KUKA KRL program: MyProgram_020().src

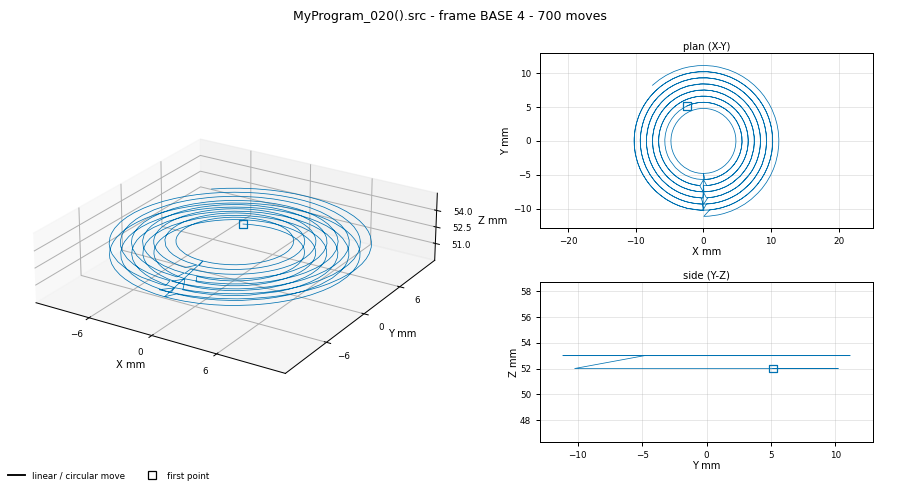
[picture p0: tool path of MyProgram_020().src in frame BASE 4, 700 of 700 moves have a stored position in this frame; points joined in program order, loops and branches not executed]
&ACCESS RVP
&REL 1
&PARAM TEMPLATE = C:\KRC\Roboter\Template\vorgabe
&PARAM EDITMASK = *
DEF MyProgram_020()
; ---- Setting reference (Base) ----
$BASE = BASE_DATA[4]

; --------------------------
; ---- Setting tool (TCP) ----
$TOOL = TOOL_DATA[3]
; --------------------------

$VEL.CP = VEL_APROX_PRINT
Startdeposition()
$VEL.CP = VEL_PRINT
LIN {X -2.4289,Y 5.1735,Z 52,A 107.8643,B 7.4449,C -0.6413,E1 7.4115,E2 338.3132} C_DIS
LIN {X -1.6441,Y 5.4719,Z 52,A 99.8653,B 7.4442,C -0.6489,E1 7.4326,E2 346.3058} C_DIS
LIN {X -0.8249,Y 5.6543,Z 52,A 90.902,B 7.4438,C -0.6532,E1 7.4572,E2 355.2666} C_DIS
LIN {X 0.0125,Y 5.7128,Z 52,A 82.6554,B 7.4438,C -0.654,E1 7.4801,E2 363.5085} C_DIS
LIN {X 0.8493,Y 5.6486,Z 52,A 74.2833,B 7.444,C -0.6514,E1 7.5034,E2 371.877} C_DIS
LIN {X 1.6675,Y 5.4622,Z 52,A 66.0095,B 7.4445,C -0.6455,E1 7.5257,E2 380.1475} C_DIS
LIN {X 2.45,Y 5.1592,Z 52,A 57.6846,B 7.4453,C -0.6363,E1 7.547,E2 388.4701} C_DIS
LIN {X 3.1799,Y 4.7453,Z 52,A 49.0733,B 7.4464,C -0.6235,E1 7.5674,E2 397.0811} C_DIS
LIN {X 3.84,Y 4.2269,Z 52,A 40.9883,B 7.4475,C -0.6091,E1 7.5847,E2 405.1642} C_DIS
LIN {X 4.4185,Y 3.6191,Z 52,A 32.7931,B 7.4489,C -0.5921,E1 7.5998,E2 413.359} C_DIS
LIN {X 4.9013,Y 2.9327,Z 52,A 24.252,B 7.4505,C -0.5719,E1 7.6128,E2 421.9018} C_DIS
LIN {X 5.2775,Y 2.1826,Z 52,A 16.2305,B 7.452,C -0.5517,E1 7.6221,E2 429.9236} C_DIS
LIN {X 5.5407,Y 1.3859,Z 52,A 7.7366,B 7.4536,C -0.5287,E1 7.6287,E2 438.4207} C_DIS
LIN {X 5.6841,Y 0.559,Z 52,A -0.2052,B 7.4552,C -0.5068,E1 7.6317,E2 446.3637} C_DIS
LIN {X 5.7063,Y -0.2799,Z 52,A -8.637,B 7.4567,C -0.483,E1 7.6315,E2 454.7997} C_DIS
LIN {X 5.6052,Y -1.1134,Z 52,A -14.4105,B 7.4577,C -0.4683,E1 7.6293,E2 460.5652} C_DIS
LIN {X 5.3986,Y -1.8885,Z 52,A -25.028,B 7.4595,C -0.4378,E1 7.621,E2 471.1999} C_DIS
LIN {X 5.0036,Y -2.7563,Z 52,A -33.9588,B 7.4608,C -0.4152,E1 7.61,E2 480.1335} C_DIS
LIN {X 4.593,Y -3.3992,Z 52,A -41.3661,B 7.4617,C -0.3977,E1 7.5983,E2 487.5447} C_DIS
LIN {X 4.0994,Y -3.9806,Z 52,A -49.0567,B 7.4626,C -0.3811,E1 7.5839,E2 495.2405} C_DIS
LIN {X 3.5319,Y -4.4901,Z 52,A -56.3617,B 7.4633,C -0.3674,E1 7.5683,E2 502.5489} C_DIS
LIN {X 2.9036,Y -4.9227,Z 52,A -64.2388,B 7.4639,C -0.3545,E1 7.5497,E2 510.4321} C_DIS
LIN {X 2.0463,Y -5.3406,Z 52,A -74.1091,B 7.4645,C -0.3422,E1 7.5245,E2 520.3099} C_DIS
LIN {X 1.0479,Y -5.6234,Z 52,A -84.1452,B 7.4648,C -0.3346,E1 7.4972,E2 530.3501} C_DIS
LIN {X 0.0063,Y -5.7151,Z 52,A -91.1459,B 7.4648,C -0.334,E1 7.4778,E2 537.3392} C_DIS
Enddeposition()
LIN {X 0.0063,Y -5.7151,Z 52,A -91.1459,B 7.4648,C -0.334,E1 7.4778,E2 537.3392} C_DIS
Startdeposition()
$VEL.CP = VEL_PRINT
LIN {X 0.5059,Y -6.5997,Z 52,A -88.5846,B 14.3606,C -1.1497,E1 14.4231,E2 533.3207} C_DIS
LIN {X 1.2106,Y -6.5077,Z 52,A -82.7819,B 14.3603,C -1.1527,E1 14.4391,E2 527.5162} C_DIS
LIN {X 1.9017,Y -6.3422,Z 52,A -76.5011,B 14.3599,C -1.1585,E1 14.456,E2 521.2307} C_DIS
LIN {X 2.57,Y -6.1008,Z 52,A -70.0036,B 14.3592,C -1.1667,E1 14.4729,E2 514.7265} C_DIS
LIN {X 3.2083,Y -5.7883,Z 52,A -64.1643,B 14.3586,C -1.175,E1 14.4874,E2 508.884} C_DIS
LIN {X 3.8105,Y -5.411,Z 52,A -58.3414,B 14.3578,C -1.1846,E1 14.5009,E2 503.0578} C_DIS
LIN {X 4.3704,Y -4.9735,Z 52,A -51.9483,B 14.3567,C -1.1974,E1 14.5147,E2 496.6579} C_DIS
LIN {X 4.8775,Y -4.4757,Z 52,A -45.8563,B 14.3557,C -1.2106,E1 14.5265,E2 490.5605} C_DIS
LIN {X 5.3296,Y -3.9273,Z 52,A -39.7457,B 14.3545,C -1.2251,E1 14.537,E2 484.4443} C_DIS
LIN {X 5.7197,Y -3.3333,Z 52,A -33.6906,B 14.3532,C -1.2403,E1 14.5459,E2 478.3839} C_DIS
LIN {X 6.0441,Y -2.7011,Z 52,A -27.6738,B 14.3518,C -1.2562,E1 14.5532,E2 472.3621} C_DIS
LIN {X 6.2999,Y -2.038,Z 52,A -21.6099,B 14.3504,C -1.2729,E1 14.5588,E2 466.2929} C_DIS
LIN {X 6.4828,Y -1.3513,Z 52,A -15.3375,B 14.3488,C -1.291,E1 14.5629,E2 460.0143} C_DIS
LIN {X 6.5887,Y -0.6485,Z 52,A -9.1544,B 14.3472,C -1.3089,E1 14.565,E2 453.8255} C_DIS
LIN {X 6.6197,Y 0.0616,Z 52,A -3.3981,B 14.3457,C -1.3251,E1 14.5652,E2 448.0663} C_DIS
LIN {X 6.575,Y 0.7709,Z 52,A 2.9779,B 14.3441,C -1.3437,E1 14.5636,E2 441.6843} C_DIS
LIN {X 6.4526,Y 1.4709,Z 52,A 8.8677,B 14.3426,C -1.36,E1 14.5604,E2 435.7915} C_DIS
LIN {X 6.2583,Y 2.1544,Z 52,A 14.9851,B 14.341,C -1.3766,E1 14.5552,E2 429.6704} C_DIS
LIN {X 5.9913,Y 2.8129,Z 52,A 21.1227,B 14.3395,C -1.3927,E1 14.5484,E2 423.5294} C_DIS
LIN {X 5.6548,Y 3.4389,Z 52,A 27.1939,B 14.3381,C -1.4075,E1 14.5399,E2 417.4557} C_DIS
LIN {X 5.2532,Y 4.0251,Z 52,A 32.9462,B 14.3368,C -1.4202,E1 14.5306,E2 411.7031} C_DIS
LIN {X 4.7937,Y 4.5673,Z 52,A 39.7226,B 14.3354,C -1.435,E1 14.5179,E2 404.9217} C_DIS
LIN {X 4.2744,Y 5.0525,Z 52,A 45.4975,B 14.3344,C -1.4453,E1 14.5058,E2 399.1475} C_DIS
LIN {X 3.7079,Y 5.4814,Z 52,A 51.459,B 14.3335,C -1.4546,E1 14.4923,E2 393.1864} C_DIS
LIN {X 3.1001,Y 5.8495,Z 52,A 57.6669,B 14.3326,C -1.4631,E1 14.4772,E2 386.9783} C_DIS
LIN {X 2.4551,Y 6.1484,Z 52,A 63.8557,B 14.332,C -1.4697,E1 14.4613,E2 380.79} C_DIS
LIN {X 1.7816,Y 6.3754,Z 52,A 70.1248,B 14.3315,C -1.4746,E1 14.4446,E2 374.5216} C_DIS
LIN {X 1.0876,Y 6.5283,Z 52,A 76.1758,B 14.3312,C -1.4773,E1 14.428,E2 368.473} C_DIS
LIN {X 0.3815,Y 6.6083,Z 52,A 82.1093,B 14.3312,C -1.478,E1 14.4115,E2 362.543} C_DIS
LIN {X -0.3292,Y 6.612,Z 52,A 88.3773,B 14.3312,C -1.4772,E1 14.3941,E2 356.2775} C_DIS
LIN {X -1.0362,Y 6.5401,Z 52,A 94.7434,B 14.3315,C -1.4745,E1 14.3765,E2 349.914} C_DIS
LIN {X -1.7309,Y 6.3897,Z 52,A 100.697,B 14.332,C -1.4697,E1 14.3603,E2 343.9653} C_DIS
LIN {X -2.406,Y 6.1677,Z 52,A 106.9909,B 14.3326,C -1.4632,E1 14.3438,E2 337.6751} C_DIS
LIN {X -3.0531,Y 5.874,Z 52,A 113.1471,B 14.3334,C -1.4549,E1 14.3284,E2 331.5237} C_DIS
LIN {X -3.6652,Y 5.513,Z 52,A 119.5582,B 14.3344,C -1.4448,E1 14.3132,E2 325.1167} C_DIS
LIN {X -4.2335,Y 5.0864,Z 52,A 125.4069,B 14.3355,C -1.4336,E1 14.3004,E2 319.2746} C_DIS
LIN {X -4.7554,Y 4.6042,Z 52,A 131.6596,B 14.3368,C -1.4206,E1 14.2879,E2 313.0271} C_DIS
LIN {X -5.2215,Y 4.0678,Z 52,A 138.0783,B 14.3382,C -1.4062,E1 14.2766,E2 306.6131} C_DIS
LIN {X -5.6279,Y 3.4848,Z 52,A 143.9789,B 14.3396,C -1.3913,E1 14.2675,E2 300.7194} C_DIS
LIN {X -5.9707,Y 2.8622,Z 52,A 150.3688,B 14.3412,C -1.3749,E1 14.2594,E2 294.3344} C_DIS
LIN {X -6.2429,Y 2.2057,Z 52,A 156.6547,B 14.3428,C -1.3578,E1 14.2531,E2 288.0535} C_DIS
LIN {X -6.443,Y 1.5238,Z 52,A 162.8172,B 14.3444,C -1.3404,E1 14.2487,E2 281.8967} C_DIS
LIN {X -6.5695,Y 0.8245,Z 52,A 169.0218,B 14.346,C -1.3226,E1 14.2461,E2 275.6972} C_DIS
LIN {X -6.6205,Y 0.1156,Z 52,A 175.3298,B 14.3476,C -1.3045,E1 14.2453,E2 269.3938} C_DIS
LIN {X -6.5942,Y -0.5946,Z 52,A -178.5062,B 14.3492,C -1.2868,E1 14.2464,E2 263.2346} C_DIS
LIN {X -6.493,Y -1.2981,Z 52,A -172.1603,B 14.3507,C -1.2691,E1 14.2494,E2 256.8923} C_DIS
LIN {X -6.3143,Y -1.9859,Z 52,A -165.8812,B 14.3522,C -1.252,E1 14.2543,E2 250.6166} C_DIS
LIN {X -6.0635,Y -2.6508,Z 52,A -159.9404,B 14.3535,C -1.2361,E1 14.2605,E2 244.6802} C_DIS
LIN {X -5.7462,Y -3.2866,Z 52,A -153.5703,B 14.3548,C -1.2205,E1 14.2689,E2 238.3123} C_DIS
LIN {X -5.3603,Y -3.8833,Z 52,A -147.4437,B 14.356,C -1.2063,E1 14.2786,E2 232.1883} C_DIS
LIN {X -4.9136,Y -4.4361,Z 52,A -141.2576,B 14.3571,C -1.1932,E1 14.2898,E2 226.004} C_DIS
LIN {X -4.4101,Y -4.9378,Z 52,A -134.9577,B 14.358,C -1.1815,E1 14.3026,E2 219.7047} C_DIS
LIN {X -3.8554,Y -5.382,Z 52,A -128.8622,B 14.3588,C -1.1715,E1 14.3162,E2 213.6102} C_DIS
LIN {X -3.2567,Y -5.7648,Z 52,A -122.6586,B 14.3595,C -1.163,E1 14.331,E2 207.4065} C_DIS
LIN {X -2.6196,Y -6.0793,Z 52,A -116.4199,B 14.36,C -1.1564,E1 14.3468,E2 201.1667} C_DIS
LIN {X -1.9529,Y -6.3257,Z 52,A -110.0034,B 14.3604,C -1.1517,E1 14.3638,E2 194.7477} C_DIS
LIN {X -1.2629,Y -6.4961,Z 52,A -104.1246,B 14.3606,C -1.1486,E1 14.3798,E2 188.8685} C_DIS
LIN {X -0.5594,Y -6.5953,Z 52,A -98.0781,B 14.3607,C -1.1473,E1 14.3966,E2 182.8202} C_DIS
LIN {X -0.5594,Y -6.5953,Z 52,A -98.0781,B 14.3607,C -1.1473,E1 14.3966,E2 182.8202} C_DIS
Enddeposition()
LIN {X -0.0274,Y -7.5244,Z 52,A -96.5126,B 21.2617,C -2.355,E1 21.386,E2 179.6143} C_DIS
Startdeposition()
$VEL.CP = VEL_PRINT
LIN {X -0.7814,Y -7.4872,Z 52,A -104.2237,B 21.2622,C -2.351,E1 21.3645,E2 187.3398} C_DIS
LIN {X -1.7575,Y -7.3207,Z 52,A -111.969,B 21.2619,C -2.3537,E1 21.3433,E2 195.0882} C_DIS
LIN {X -2.7152,Y -7.0156,Z 52,A -119.2275,B 21.2612,C -2.3604,E1 21.3242,E2 202.3448} C_DIS
LIN {X -3.4481,Y -6.6852,Z 52,A -125.2958,B 21.2604,C -2.3675,E1 21.309,E2 208.4122} C_DIS
LIN {X -4.1421,Y -6.2795,Z 52,A -131.442,B 21.2595,C -2.3762,E1 21.2944,E2 214.5574} C_DIS
LIN {X -4.7888,Y -5.8017,Z 52,A -137.6042,B 21.2584,C -2.3866,E1 21.2808,E2 220.7177} C_DIS
LIN {X -5.3803,Y -5.2573,Z 52,A -143.6754,B 21.2571,C -2.3986,E1 21.2687,E2 226.7856} C_DIS
LIN {X -6.0374,Y -4.4969,Z 52,A -151.9759,B 21.2552,C -2.4157,E1 21.2541,E2 235.0848} C_DIS
LIN {X -6.6618,Y -3.4963,Z 52,A -160.598,B 21.2528,C -2.4381,E1 21.242,E2 243.698} C_DIS
LIN {X -7.1224,Y -2.4411,Z 52,A -170.0178,B 21.2501,C -2.4625,E1 21.2324,E2 253.1129} C_DIS
LIN {X -7.3822,Y -1.4736,Z 52,A -177.4448,B 21.2477,C -2.4844,E1 21.2277,E2 260.5309} C_DIS
LIN {X -7.5117,Y -0.49,Z 52,A 175.1182,B 21.2452,C -2.5068,E1 21.2256,E2 267.9588} C_DIS
LIN {X -7.5011,Y 0.6008,Z 52,A 168.4839,B 21.2425,C -2.5302,E1 21.226,E2 274.5756} C_DIS
LIN {X -7.3321,Y 1.704,Z 52,A 157.0482,B 21.2393,C -2.5585,E1 21.2317,E2 286.0133} C_DIS
LIN {X -6.9123,Y 2.9745,Z 52,A 148.1141,B 21.236,C -2.5868,E1 21.2403,E2 294.929} C_DIS
LIN {X -6.3173,Y 4.0959,Z 52,A 138.4221,B 21.233,C -2.6128,E1 21.2537,E2 304.609} C_DIS
LIN {X -5.7816,Y 4.8207,Z 52,A 131.1882,B 21.2309,C -2.63,E1 21.2661,E2 311.8358} C_DIS
LIN {X -4.9317,Y 5.6867,Z 52,A 121.5646,B 21.2285,C -2.6503,E1 21.2855,E2 321.4502} C_DIS
LIN {X -3.9768,Y 6.3909,Z 52,A 112.154,B 21.2266,C -2.6668,E1 21.3072,E2 330.8528} C_DIS
LIN {X -3.1751,Y 6.826,Z 52,A 104.5371,B 21.2254,C -2.6765,E1 21.3263,E2 338.4661} C_DIS
LIN {X -1.7524,Y 7.3221,Z 52,A 94.415,B 21.2238,C -2.6895,E1 21.3533,E2 348.5726} C_DIS
LIN {X -0.7984,Y 7.4853,Z 52,A 87.1848,B 21.2233,C -2.694,E1 21.3732,E2 355.7973} C_DIS
LIN {X 0.1483,Y 7.5262,Z 52,A 79.6626,B 21.2232,C -2.6949,E1 21.3942,E2 363.3174} C_DIS
LIN {X 1.1941,Y 7.4322,Z 52,A 71.8258,B 21.2233,C -2.6936,E1 21.4159,E2 371.1506} C_DIS
LIN {X 2.1413,Y 7.2172,Z 52,A 64.1331,B 21.224,C -2.6884,E1 21.4367,E2 378.8437} C_DIS
LIN {X 3.0246,Y 6.8934,Z 52,A 56.7749,B 21.2249,C -2.6807,E1 21.4557,E2 386.2029} C_DIS
LIN {X 4.1385,Y 6.2822,Z 52,A 47.6638,B 21.2263,C -2.6693,E1 21.4776,E2 395.3123} C_DIS
LIN {X 4.7085,Y 5.8745,Z 52,A 41.823,B 21.2276,C -2.6581,E1 21.4905,E2 401.1581} C_DIS
LIN {X 5.57,Y 5.0582,Z 52,A 33.2892,B 21.2295,C -2.642,E1 21.5073,E2 409.6932} C_DIS
LIN {X 6.1111,Y 4.3879,Z 52,A 26.9308,B 21.2312,C -2.6278,E1 21.5181,E2 416.0546} C_DIS
LIN {X 6.715,Y 3.4036,Z 52,A 17.7733,B 21.234,C -2.6038,E1 21.5307,E2 425.2216} C_DIS
LIN {X 7.1416,Y 2.3681,Z 52,A 11.3801,B 21.2356,C -2.5907,E1 21.5373,E2 431.6086} C_DIS
LIN {X 7.3518,Y 1.6184,Z 52,A 3.4647,B 21.2387,C -2.5638,E1 21.5428,E2 439.5435} C_DIS
LIN {X 7.5047,Y 0.5929,Z 52,A -4.3405,B 21.2413,C -2.5408,E1 21.5454,E2 447.3571} C_DIS
LIN {X 7.5175,Y -0.4036,Z 52,A -11.7653,B 21.2438,C -2.5187,E1 21.545,E2 454.7899} C_DIS
LIN {X 7.4202,Y -1.2685,Z 52,A -19.3373,B 21.2466,C -2.494,E1 21.5418,E2 462.3766} C_DIS
LIN {X 7.0514,Y -2.6343,Z 52,A -28.9248,B 21.2495,C -2.4683,E1 21.5338,E2 471.9698} C_DIS
LIN {X 6.7153,Y -3.403,Z 52,A -35.7286,B 21.2517,C -2.4483,E1 21.5256,E2 478.7848} C_DIS
LIN {X 6.1358,Y -4.3568,Z 52,A -42.0446,B 21.253,C -2.4361,E1 21.5162,E2 485.0964} C_DIS
LIN {X 5.4535,Y -5.1882,Z 52,A -53.8238,B 21.2569,C -2.4006,E1 21.4945,E2 496.9101} C_DIS
LIN {X 4.3237,Y -6.1617,Z 52,A -63.1188,B 21.2584,C -2.386,E1 21.4741,E2 506.2042} C_DIS
LIN {X 3.4446,Y -6.6892,Z 52,A -70.8047,B 21.2598,C -2.3735,E1 21.4555,E2 513.8971} C_DIS
LIN {X 2.4008,Y -7.136,Z 52,A -79.8175,B 21.2611,C -2.3612,E1 21.432,E2 522.9202} C_DIS
LIN {X 1.5119,Y -7.3741,Z 52,A -86.7893,B 21.2617,C -2.3551,E1 21.413,E2 529.897} C_DIS
LIN {X 0.7619,Y -7.4894,Z 52,A -92.7274,B 21.2621,C -2.3515,E1 21.3966,E2 535.8397} C_DIS
LIN {X -0.0274,Y -7.5244,Z 52,A -96.5127,B 21.2617,C -2.355,E1 21.386,E2 539.6144} C_DIS
Enddeposition()
LIN {X -0.0274,Y -7.5244,Z 52,A -96.5127,B 21.2617,C -2.355,E1 21.386,E2 539.6144} C_DIS
Startdeposition()
$VEL.CP = VEL_PRINT
LIN {X 0.4505,Y -8.4164,Z 52,A -93.4741,B 24.8134,C -3.1503,E1 25.0114,E2 535.6406} C_DIS
LIN {X 1.5174,Y -8.2959,Z 52,A -85.4803,B 24.8125,C -3.1575,E1 25.0336,E2 527.6369} C_DIS
LIN {X 2.6389,Y -8.0045,Z 52,A -77.6649,B 24.8115,C -3.1657,E1 25.0546,E2 519.8149} C_DIS
LIN {X 3.713,Y -7.57,Z 52,A -69.6264,B 24.8101,C -3.1779,E1 25.0751,E2 511.7673} C_DIS
LIN {X 4.7012,Y -7.0001,Z 52,A -62.0699,B 24.8085,C -3.1911,E1 25.093,E2 504.2033} C_DIS
LIN {X 5.435,Y -6.4462,Z 52,A -53.1824,B 24.8052,C -3.2179,E1 25.1121,E2 495.2863} C_DIS
LIN {X 7.0088,Y -4.6885,Z 52,A -40.2537,B 24.8023,C -3.2418,E1 25.1348,E2 482.361} C_DIS
LIN {X 7.4731,Y -3.9082,Z 52,A -33.7544,B 24.8,C -3.2609,E1 25.1437,E2 475.8499} C_DIS
LIN {X 7.8918,Y -2.9691,Z 52,A -26.4626,B 24.7972,C -3.2833,E1 25.1514,E2 468.5453} C_DIS
LIN {X 8.222,Y -1.8731,Z 52,A -18.8386,B 24.7944,C -3.3061,E1 25.1569,E2 460.9111} C_DIS
LIN {X 8.3909,Y -0.8376,Z 52,A -12.2741,B 24.792,C -3.3249,E1 25.1593,E2 454.3408} C_DIS
LIN {X 8.4309,Y 0.142,Z 52,A -5.498,B 24.7893,C -3.3462,E1 25.1596,E2 447.5544} C_DIS
LIN {X 8.3647,Y 1.0691,Z 52,A 1.2925,B 24.7865,C -3.3683,E1 25.1577,E2 440.7516} C_DIS
LIN {X 8.1134,Y 2.2842,Z 52,A 9.2044,B 24.7837,C -3.3904,E1 25.1526,E2 432.8332} C_DIS
LIN {X 7.7187,Y 3.3947,Z 52,A 17.3327,B 24.7807,C -3.4135,E1 25.1443,E2 424.6951} C_DIS
LIN {X 7.2312,Y 4.3372,Z 52,A 24.5613,B 24.7783,C -3.4324,E1 25.1345,E2 417.4593} C_DIS
LIN {X 6.6288,Y 5.2057,Z 52,A 31.6279,B 24.7761,C -3.4489,E1 25.1228,E2 410.3876} C_DIS
LIN {X 6.0725,Y 5.8426,Z 52,A 37.0713,B 24.7747,C -3.4598,E1 25.1126,E2 404.9424} C_DIS
LIN {X 5.4563,Y 6.4214,Z 52,A 42.825,B 24.7733,C -3.4708,E1 25.1006,E2 399.1853} C_DIS
LIN {X 4.6138,Y 7.0597,Z 52,A 50.4541,B 24.7715,C -3.4843,E1 25.0831,E2 391.5506} C_DIS
LIN {X 3.5901,Y 7.625,Z 52,A 57.9991,B 24.7704,C -3.4927,E1 25.0645,E2 384.0065} C_DIS
LIN {X 2.785,Y 7.9551,Z 52,A 63.8459,B 24.7697,C -3.4978,E1 25.0492,E2 378.1601} C_DIS
LIN {X 1.95,Y 8.1997,Z 52,A 69.7666,B 24.7692,C -3.5015,E1 25.0332,E2 372.24} C_DIS
LIN {X 0.7662,Y 8.3987,Z 52,A 78.3807,B 24.7688,C -3.5045,E1 25.0094,E2 363.6258} C_DIS
LIN {X -0.4208,Y 8.4227,Z 52,A 87.5718,B 24.7687,C -3.5053,E1 24.9838,E2 354.432} C_DIS
LIN {X -2.3301,Y 8.1054,Z 52,A 99.4928,B 24.7705,C -3.492,E1 24.9513,E2 342.5286} C_DIS
LIN {X -3.4977,Y 7.6741,Z 52,A 108.1812,B 24.7719,C -3.4809,E1 24.9289,E2 333.8473} C_DIS
LIN {X -4.5027,Y 7.1259,Z 52,A 115.3498,B 24.7737,C -3.467,E1 24.9116,E2 326.6906} C_DIS
LIN {X -5.4177,Y 6.461,Z 52,A 123.1877,B 24.7758,C -3.4514,E1 24.8942,E2 318.8616} C_DIS
LIN {X -6.1286,Y 5.7846,Z 52,A 129.6137,B 24.7778,C -3.436,E1 24.8815,E2 312.4455} C_DIS
LIN {X -6.8592,Y 4.9051,Z 52,A 137.784,B 24.7804,C -3.4162,E1 24.8674,E2 304.2843} C_DIS
LIN {X -7.5549,Y 3.7442,Z 52,A 147.3187,B 24.7837,C -3.3905,E1 24.8544,E2 294.7612} C_DIS
LIN {X -8.127,Y 2.2469,Z 52,A 160.9266,B 24.7879,C -3.3573,E1 24.8428,E2 281.1551} C_DIS
LIN {X -8.4128,Y 0.5678,Z 52,A 169.886,B 24.7924,C -3.3222,E1 24.8399,E2 272.2265} C_DIS
LIN {X -8.4247,Y -0.3871,Z 52,A 176.7329,B 24.7949,C -3.302,E1 24.8403,E2 265.3867} C_DIS
LIN {X -8.2786,Y -1.5841,Z 52,A -176.9993,B 24.7979,C -3.2777,E1 24.8426,E2 259.1397} C_DIS
LIN {X -8.1045,Y -2.3329,Z 52,A -169.8712,B 24.7999,C -3.2619,E1 24.8476,E2 252.008} C_DIS
LIN {X -7.751,Y -3.3079,Z 52,A -163.2341,B 24.8023,C -3.2422,E1 24.8542,E2 245.3808} C_DIS
LIN {X -7.3886,Y -4.054,Z 52,A -157.4386,B 24.8041,C -3.2273,E1 24.8617,E2 239.5901} C_DIS
LIN {X -6.8394,Y -4.9337,Z 52,A -149.9463,B 24.8062,C -3.2101,E1 24.8733,E2 232.1017} C_DIS
LIN {X -6.1425,Y -5.7759,Z 52,A -142.8279,B 24.8082,C -3.1937,E1 24.8864,E2 224.9904} C_DIS
LIN {X -5.3899,Y -6.4771,Z 52,A -136.0085,B 24.8098,C -3.1804,E1 24.9006,E2 218.1758} C_DIS
LIN {X -4.5644,Y -7.0908,Z 52,A -128.4213,B 24.811,C -3.1699,E1 24.918,E2 210.5878} C_DIS
LIN {X -3.6707,Y -7.5906,Z 52,A -121.6991,B 24.8121,C -3.161,E1 24.9346,E2 203.8685} C_DIS
LIN {X -2.7148,Y -7.9848,Z 52,A -114.2313,B 24.8127,C -3.1557,E1 24.9542,E2 196.3979} C_DIS
LIN {X -1.5311,Y -8.2879,Z 52,A -106.4733,B 24.8133,C -3.1506,E1 24.9753,E2 188.6421} C_DIS
LIN {X -0.3286,Y -8.4268,Z 52,A -98.0691,B 24.8133,C -3.1508,E1 24.9986,E2 180.2337} C_DIS
LIN {X -0.3286,Y -8.4268,Z 52,A -98.0691,B 24.8133,C -3.1508,E1 24.9986,E2 180.2337} C_DIS
Enddeposition()
LIN {X -0.052,Y -9.3359,Z 52,A -98.3791,B 24.8159,C -3.1288,E1 24.9976,E2 180.5961} C_DIS
Startdeposition()
$VEL.CP = VEL_PRINT
LIN {X -0.8395,Y -9.3001,Z 52,A -104.3026,B 24.8163,C -3.1254,E1 24.9811,E2 186.5298} C_DIS
LIN {X -1.9855,Y -9.1183,Z 52,A -111.0179,B 24.8159,C -3.1289,E1 24.9627,E2 193.2436} C_DIS
LIN {X -2.7999,Y -8.9013,Z 52,A -116.1132,B 24.8155,C -3.1324,E1 24.949,E2 198.3387} C_DIS
LIN {X -3.5922,Y -8.6137,Z 52,A -121.2417,B 24.8149,C -3.1372,E1 24.9357,E2 203.4669} C_DIS
LIN {X -4.6382,Y -8.1037,Z 52,A -128.6231,B 24.814,C -3.1455,E1 24.9174,E2 210.8486} C_DIS
LIN {X -5.456,Y -7.5777,Z 52,A -134.7044,B 24.8129,C -3.1546,E1 24.9033,E2 216.9285} C_DIS
LIN {X -6.282,Y -6.9086,Z 52,A -142.2,B 24.8115,C -3.1658,E1 24.8875,E2 224.4268} C_DIS
LIN {X -7.0554,Y -6.1139,Z 52,A -148.6364,B 24.8097,C -3.1807,E1 24.8755,E2 230.856} C_DIS
LIN {X -7.8689,Y -5.0191,Z 52,A -156.4687,B 24.8073,C -3.2012,E1 24.863,E2 238.6777} C_DIS
LIN {X -8.4491,Y -3.9729,Z 52,A -163.7812,B 24.8049,C -3.2206,E1 24.8535,E2 245.9827} C_DIS
LIN {X -8.7989,Y -3.1225,Z 52,A -169.5115,B 24.803,C -3.2364,E1 24.8478,E2 251.7073} C_DIS
LIN {X -9.0977,Y -2.0829,Z 52,A -176.1379,B 24.8006,C -3.256,E1 24.8431,E2 258.3253} C_DIS
LIN {X -9.2807,Y -1.0169,Z 52,A 177.0006,B 24.7981,C -3.2761,E1 24.8403,E2 265.1795} C_DIS
LIN {X -9.3371,Y 0.0703,Z 52,A 169.9229,B 24.7955,C -3.2968,E1 24.8399,E2 272.2501} C_DIS
LIN {X -9.269,Y 1.1202,Z 52,A 162.711,B 24.793,C -3.317,E1 24.8419,E2 279.4569} C_DIS
LIN {X -8.9578,Y 2.6352,Z 52,A 154.006,B 24.7894,C -3.3458,E1 24.8477,E2 288.1436} C_DIS
LIN {X -8.5926,Y 3.6417,Z 52,A 147.8018,B 24.7869,C -3.3653,E1 24.8539,E2 294.3359} C_DIS
LIN {X -8.1226,Y 4.6038,Z 52,A 140.5918,B 24.7845,C -3.3838,E1 24.8633,E2 301.5399} C_DIS
LIN {X -7.3654,Y 5.7368,Z 52,A 132.4678,B 24.7817,C -3.4059,E1 24.8764,E2 309.6507} C_DIS
LIN {X -6.6986,Y 6.5035,Z 52,A 126.1589,B 24.7798,C -3.4209,E1 24.8883,E2 315.9515} C_DIS
LIN {X -5.7812,Y 7.3262,Z 52,A 118.7773,B 24.7776,C -3.4374,E1 24.9039,E2 323.3221} C_DIS
LIN {X -5.0269,Y 7.8637,Z 52,A 112.9356,B 24.7762,C -3.448,E1 24.9174,E2 329.158} C_DIS
LIN {X -4.016,Y 8.4282,Z 52,A 105.736,B 24.7748,C -3.4592,E1 24.9352,E2 336.3506} C_DIS
LIN {X -2.9275,Y 8.8627,Z 52,A 98.7091,B 24.7735,C -3.4686,E1 24.9535,E2 343.3694} C_DIS
LIN {X -1.7907,Y 9.1636,Z 52,A 91.1938,B 24.7728,C -3.4744,E1 24.9739,E2 350.8809} C_DIS
LIN {X -0.6773,Y 9.3118,Z 52,A 84.2906,B 24.7723,C -3.4779,E1 24.9931,E2 357.7797} C_DIS
LIN {X 0.6229,Y 9.3154,Z 52,A 76.4024,B 24.7722,C -3.4791,E1 25.0151,E2 365.6637} C_DIS
LIN {X 1.7844,Y 9.1611,Z 52,A 69.2149,B 24.7724,C -3.4771,E1 25.0349,E2 372.849} C_DIS
LIN {X 2.6524,Y 8.9468,Z 52,A 63.9703,B 24.7728,C -3.4746,E1 25.049,E2 378.0913} C_DIS
LIN {X 3.7043,Y 8.5697,Z 52,A 56.8714,B 24.7737,C -3.4671,E1 25.0675,E2 385.1923} C_DIS
LIN {X 4.7988,Y 8.0048,Z 52,A 50.9112,B 24.7741,C -3.4643,E1 25.0822,E2 391.1423} C_DIS
LIN {X 5.4668,Y 7.5701,Z 52,A 44.5238,B 24.776,C -3.4498,E1 25.097,E2 397.5428} C_DIS
LIN {X 6.1655,Y 7.0114,Z 52,A 38.9428,B 24.7774,C -3.4392,E1 25.1089,E2 403.1274} C_DIS
LIN {X 7.152,Y 6.0011,Z 52,A 30.3335,B 24.7797,C -3.421,E1 25.1252,E2 411.7421} C_DIS
LIN {X 7.7543,Y 5.2005,Z 52,A 24.2516,B 24.7816,C -3.4066,E1 25.1351,E2 417.8287} C_DIS
LIN {X 8.3413,Y 4.186,Z 52,A 17.2885,B 24.7839,C -3.3891,E1 25.1445,E2 424.7969} C_DIS
LIN {X 8.8069,Y 3.1008,Z 52,A 10.0363,B 24.7865,C -3.3687,E1 25.1519,E2 432.0574} C_DIS
LIN {X 9.0454,Y 2.3117,Z 52,A 4.8737,B 24.7884,C -3.3533,E1 25.1558,E2 437.2269} C_DIS
LIN {X 9.2553,Y 1.2386,Z 52,A -3.0125,B 24.7919,C -3.326,E1 25.1592,E2 445.1317} C_DIS
LIN {X 9.3328,Y -0.2628,Z 52,A -10.8383,B 24.7944,C -3.3059,E1 25.1596,E2 452.9586} C_DIS
LIN {X 9.1482,Y -1.8645,Z 52,A -22.7728,B 24.7997,C -3.2631,E1 25.1543,E2 464.9245} C_DIS
LIN {X 8.6526,Y -3.5093,Z 52,A -31.0236,B 24.8019,C -3.245,E1 25.1468,E2 473.1717} C_DIS
LIN {X 8.0666,Y -4.704,Z 52,A -40.3815,B 24.8056,C -3.215,E1 25.1345,E2 482.5516} C_DIS
LIN {X 7.3945,Y -5.6982,Z 52,A -45.3651,B 24.8064,C -3.2088,E1 25.1265,E2 487.5255} C_DIS
LIN {X 6.7537,Y -6.4454,Z 52,A -54.3373,B 24.81,C -3.1782,E1 25.1096,E2 496.5306} C_DIS
LIN {X 5.4355,Y -7.5868,Z 52,A -61.872,B 24.8108,C -3.1716,E1 25.0934,E2 504.0525} C_DIS
LIN {X 4.8099,Y -8.0022,Z 52,A -68.0282,B 24.8128,C -3.1554,E1 25.0789,E2 510.2271} C_DIS
LIN {X 3.7305,Y -8.5544,Z 52,A -75.1902,B 24.814,C -3.1452,E1 25.0609,E2 517.3946} C_DIS
LIN {X 2.6834,Y -8.9427,Z 52,A -82.1917,B 24.8151,C -3.1362,E1 25.0423,E2 524.4037} C_DIS
LIN {X 1.6599,Y -9.189,Z 52,A -89.4964,B 24.8161,C -3.1275,E1 25.0223,E2 531.7201} C_DIS
LIN {X 0.4404,Y -9.323,Z 52,A -95.5715,B 24.8159,C -3.1289,E1 25.0055,E2 537.7885} C_DIS
LIN {X 0.4404,Y -9.323,Z 52,A -95.5715,B 24.8159,C -3.1289,E1 25.0055,E2 537.7885} C_DIS
Enddeposition()
LIN {X -0.0612,Y -10.2374,Z 52,A -97.9695,B 24.8176,C -3.1145,E1 24.9987,E2 540.2205} C_DIS
Startdeposition()
$VEL.CP = VEL_PRINT
LIN {X 0.6871,Y -10.2175,Z 52,A -92.1264,B 24.8167,C -3.1221,E1 25.015,E2 534.3609} C_DIS
LIN {X 1.7113,Y -10.0968,Z 52,A -86.2358,B 24.8162,C -3.1264,E1 25.0313,E2 528.4653} C_DIS
LIN {X 2.8814,Y -9.8282,Z 52,A -79.7051,B 24.8155,C -3.1323,E1 25.049,E2 521.9307} C_DIS
LIN {X 3.9668,Y -9.4385,Z 52,A -73.3076,B 24.8145,C -3.1406,E1 25.0657,E2 515.5273} C_DIS
LIN {X 4.8,Y -9.0423,Z 52,A -68.1956,B 24.8136,C -3.1486,E1 25.0784,E2 510.4101} C_DIS
LIN {X 5.5946,Y -8.5734,Z 52,A -63.1215,B 24.8125,C -3.1576,E1 25.0905,E2 505.3309} C_DIS
LIN {X 6.6386,Y -7.7967,Z 52,A -55.8131,B 24.8107,C -3.1729,E1 25.1065,E2 498.0132} C_DIS
LIN {X 7.4442,Y -7.0269,Z 52,A -49.6235,B 24.809,C -3.1873,E1 25.1188,E2 491.8155} C_DIS
LIN {X 8.0272,Y -6.3523,Z 52,A -44.7338,B 24.8075,C -3.1993,E1 25.1275,E2 486.9197} C_DIS
LIN {X 8.5502,Y -5.6302,Z 52,A -39.831,B 24.806,C -3.2121,E1 25.1353,E2 482.0107} C_DIS
LIN {X 9.0088,Y -4.8655,Z 52,A -34.8074,B 24.8042,C -3.2263,E1 25.1423,E2 476.9794} C_DIS
LIN {X 9.4867,Y -3.8588,Z 52,A -28.3755,B 24.8018,C -3.2457,E1 25.1495,E2 470.5366} C_DIS
LIN {X 9.8799,Y -2.6852,Z 52,A -22.9596,B 24.8005,C -3.257,E1 25.1542,E2 465.1245} C_DIS
LIN {X 10.0815,Y -1.8057,Z 52,A -16.4878,B 24.7974,C -3.2817,E1 25.158,E2 458.632} C_DIS
LIN {X 10.2129,Y -0.7557,Z 52,A -10.7283,B 24.7953,C -3.2991,E1 25.1596,E2 452.8653} C_DIS
LIN {X 10.2254,Y 0.5691,Z 52,A -3.0869,B 24.7922,C -3.3235,E1 25.1592,E2 445.2115} C_DIS
LIN {X 10.0787,Y 1.7954,Z 52,A 3.5193,B 24.7898,C -3.3426,E1 25.1566,E2 438.5989} C_DIS
LIN {X 9.8779,Y 2.6862,Z 52,A 8.5254,B 24.788,C -3.357,E1 25.1532,E2 433.5875} C_DIS
LIN {X 9.5994,Y 3.5558,Z 52,A 13.4788,B 24.7862,C -3.3707,E1 25.1487,E2 428.6296} C_DIS
LIN {X 9.2459,Y 4.3976,Z 52,A 18.7553,B 24.7843,C -3.3857,E1 25.1427,E2 423.3461} C_DIS
LIN {X 8.8161,Y 5.2032,Z 52,A 23.8601,B 24.7826,C -3.399,E1 25.1357,E2 418.2363} C_DIS
LIN {X 8.3163,Y 5.9674,Z 52,A 28.8739,B 24.7811,C -3.4109,E1 25.1277,E2 413.2188} C_DIS
LIN {X 7.7514,Y 6.6846,Z 52,A 33.8719,B 24.7796,C -3.4218,E1 25.1189,E2 408.2179} C_DIS
LIN {X 7.1257,Y 7.3495,Z 52,A 38.9606,B 24.7783,C -3.4323,E1 25.1089,E2 403.1261} C_DIS
LIN {X 6.4426,Y 7.9552,Z 52,A 44.1284,B 24.777,C -3.442,E1 25.0979,E2 397.9552} C_DIS
LIN {X 5.7087,Y 8.4984,Z 52,A 49.0874,B 24.776,C -3.4496,E1 25.0866,E2 392.9954} C_DIS
LIN {X 4.9289,Y 8.9734,Z 52,A 54.4375,B 24.775,C -3.4578,E1 25.0736,E2 387.6421} C_DIS
LIN {X 4.1092,Y 9.3757,Z 52,A 59.3893,B 24.7743,C -3.4628,E1 25.0611,E2 382.6908} C_DIS
LIN {X 3.2574,Y 9.7048,Z 52,A 64.455,B 24.7737,C -3.4671,E1 25.0478,E2 377.6254} C_DIS
LIN {X 2.3798,Y 9.9572,Z 52,A 69.5483,B 24.7733,C -3.47,E1 25.034,E2 372.533} C_DIS
LIN {X 1.7092,Y 10.0972,Z 52,A 74.0055,B 24.7729,C -3.4736,E1 25.0218,E2 368.0719} C_DIS
LIN {X 0.5608,Y 10.226,Z 52,A 80.5122,B 24.7729,C -3.4741,E1 25.0037,E2 361.5674} C_DIS
LIN {X -0.8075,Y 10.2063,Z 52,A 87.6056,B 24.7734,C -3.47,E1 24.9839,E2 354.4824} C_DIS
LIN {X -1.7266,Y 10.0914,Z 52,A 92.7707,B 24.7738,C -3.4666,E1 24.9697,E2 349.321} C_DIS
LIN {X -2.6317,Y 9.8943,Z 52,A 97.9163,B 24.7744,C -3.4618,E1 24.9557,E2 344.1799} C_DIS
LIN {X -3.5154,Y 9.6167,Z 52,A 103.2031,B 24.7752,C -3.4559,E1 24.9417,E2 338.8972} C_DIS
LIN {X -4.5793,Y 9.16,Z 52,A 110.1343,B 24.7763,C -3.4471,E1 24.9242,E2 331.9696} C_DIS
LIN {X -5.7429,Y 8.4765,Z 52,A 117.3701,B 24.7782,C -3.4331,E1 24.9071,E2 324.7446} C_DIS
LIN {X -6.4701,Y 7.933,Z 52,A 122.4181,B 24.7795,C -3.4226,E1 24.896,E2 319.7032} C_DIS
LIN {X -7.147,Y 7.328,Z 52,A 127.4329,B 24.781,C -3.4111,E1 24.8858,E2 314.6955} C_DIS
LIN {X -7.7686,Y 6.6665,Z 52,A 132.5126,B 24.7826,C -3.3987,E1 24.8763,E2 309.6228} C_DIS
LIN {X -8.3291,Y 5.9525,Z 52,A 137.7579,B 24.7843,C -3.3857,E1 24.8676,E2 304.3836} C_DIS
LIN {X -8.823,Y 5.1908,Z 52,A 142.6939,B 24.7861,C -3.3717,E1 24.8603,E2 299.4558} C_DIS
LIN {X -9.2496,Y 4.3896,Z 52,A 148.0022,B 24.7879,C -3.3573,E1 24.8537,E2 294.1537} C_DIS
LIN {X -9.6005,Y 3.5524,Z 52,A 153.0549,B 24.7898,C -3.3423,E1 24.8485,E2 289.1086} C_DIS
LIN {X -9.8773,Y 2.6878,Z 52,A 158.1339,B 24.7918,C -3.3269,E1 24.8445,E2 284.037} C_DIS
LIN {X -10.0771,Y 1.8023,Z 52,A 163.2087,B 24.7937,C -3.3113,E1 24.8417,E2 278.9697} C_DIS
LIN {X -10.198,Y 0.9025,Z 52,A 168.4066,B 24.7957,C -3.2956,E1 24.8401,E2 273.7785} C_DIS
LIN {X -10.2377,Y -0.0045,Z 52,A 173.5016,B 24.7976,C -3.2799,E1 24.8398,E2 268.6905} C_DIS
LIN {X -10.1972,Y -0.9115,Z 52,A 178.6629,B 24.7996,C -3.2643,E1 24.8408,E2 263.5356} C_DIS
LIN {X -10.0758,Y -1.8112,Z 52,A -176.2118,B 24.8015,C -3.2489,E1 24.843,E2 258.4166} C_DIS
LIN {X -9.8753,Y -2.6967,Z 52,A -171.1193,B 24.8033,C -3.2339,E1 24.8465,E2 253.3303} C_DIS
LIN {X -9.5976,Y -3.561,Z 52,A -166.1323,B 24.8051,C -3.2194,E1 24.851,E2 248.3498} C_DIS
LIN {X -9.2459,Y -4.3978,Z 52,A -160.8147,B 24.8067,C -3.2056,E1 24.8571,E2 243.0361} C_DIS
LIN {X -8.8187,Y -5.1988,Z 52,A -155.6812,B 24.8083,C -3.1925,E1 24.8641,E2 237.9071} C_DIS
LIN {X -8.3224,Y -5.9589,Z 52,A -150.8905,B 24.8099,C -3.1798,E1 24.8716,E2 233.1228} C_DIS
LIN {X -7.9126,Y -6.5029,Z 52,A -146.2833,B 24.8108,C -3.172,E1 24.8797,E2 228.5131} C_DIS
LIN {X -7.1244,Y -7.356,Z 52,A -140.2253,B 24.8125,C -3.158,E1 24.8915,E2 222.4625} C_DIS
LIN {X -6.3289,Y -8.0508,Z 52,A -134.4137,B 24.8138,C -3.1471,E1 24.9039,E2 216.6547} C_DIS
LIN {X -5.3658,Y -8.721,Z 52,A -129.0602,B 24.8152,C -3.1347,E1 24.9163,E2 211.3129} C_DIS
LIN {X -4.5747,Y -9.1622,Z 52,A -122.715,B 24.8157,C -3.1309,E1 24.9319,E2 204.959} C_DIS
LIN {X -3.5253,Y -9.6126,Z 52,A -116.3267,B 24.8164,C -3.1248,E1 24.9484,E2 198.571} C_DIS
LIN {X -2.3592,Y -9.9668,Z 52,A -109.2976,B 24.8168,C -3.1212,E1 24.9673,E2 191.5396} C_DIS
LIN {X -0.9586,Y -10.1972,Z 52,A -101.2361,B 24.817,C -3.12,E1 24.9896,E2 183.4746} C_DIS
LIN {X -0.0612,Y -10.2374,Z 52,A -97.9695,B 24.8176,C -3.1145,E1 24.9987,E2 180.2205} C_DIS
Enddeposition()
LIN {X 0.0024,Y -4.8127,Z 53,A -2.8481,B 0,C 0,E1 0.1598,E2 90.0716} C_DIS
Startdeposition()
$VEL.CP = VEL_PRINT
LIN {X -0.7063,Y -4.7565,Z 53,A -2.8719,B 0,C 0,E1 0.1598,E2 90.0717} C_DIS
LIN {X -1.2627,Y -4.6392,Z 53,A -2.8873,B 0,C 0,E1 0.1598,E2 90.0717} C_DIS
LIN {X -1.9345,Y -4.4065,Z 53,A -2.9021,B 0,C 0,E1 0.1598,E2 90.0717} C_DIS
LIN {X -2.82,Y -3.8913,Z 53,A -2.9125,B 0,C 0,E1 0.1598,E2 90.0715} C_DIS
LIN {X -3.3261,Y -3.47,Z 53,A -2.9132,B 0,C 0,E1 0.1598,E2 90.0715} C_DIS
LIN {X -3.7695,Y -2.983,Z 53,A -2.9088,B 0,C 0,E1 0.1598,E2 90.0715} C_DIS
LIN {X -4.1425,Y -2.44,Z 53,A -2.8994,B 0,C 0,E1 0.1598,E2 90.0715} C_DIS
LIN {X -4.4385,Y -1.8516,Z 53,A -2.8853,B 0,C 0,E1 0.1598,E2 90.0715} C_DIS
LIN {X -4.6474,Y -1.2269,Z 53,A -2.8664,B 0,C 0,E1 0.1598,E2 90.0715} C_DIS
LIN {X -4.7739,Y -0.5805,Z 53,A -2.8436,B 0,C 0,E1 0.1598,E2 90.0715} C_DIS
LIN {X -4.8062,Y 0.0773,Z 53,A -2.8168,B 0,C 0,E1 0.1598,E2 90.0715} C_DIS
LIN {X -4.7512,Y 0.7334,Z 53,A -2.7869,B 0,C 0,E1 0.1598,E2 90.0716} C_DIS
LIN {X -4.6063,Y 1.3759,Z 53,A -2.7544,B 0,C 0,E1 0.1598,E2 90.0716} C_DIS
LIN {X -4.375,Y 1.9926,Z 53,A -2.7197,B 0,C 0,E1 0.1598,E2 90.0717} C_DIS
LIN {X -4.0617,Y 2.5718,Z 53,A -2.6836,B 0,C 0,E1 0.1598,E2 90.0718} C_DIS
LIN {X -3.6727,Y 3.1034,Z 53,A -2.6467,B 0,C 0,E1 0.1598,E2 90.0718} C_DIS
LIN {X -3.2143,Y 3.5765,Z 53,A -2.6098,B 0,C 0,E1 0.1598,E2 90.072} C_DIS
LIN {X -2.6959,Y 3.983,Z 53,A -2.5735,B 0,C 0,E1 0.1598,E2 90.072} C_DIS
LIN {X -2.1259,Y 4.3136,Z 53,A -2.5385,B 0,C 0,E1 0.1598,E2 90.0721} C_DIS
LIN {X -1.5161,Y 4.5626,Z 53,A -2.5054,B 0,C 0,E1 0.1598,E2 90.0722} C_DIS
LIN {X -0.8781,Y 4.727,Z 53,A -2.475,B 0,C 0,E1 0.1598,E2 90.0722} C_DIS
LIN {X -0.2239,Y 4.8036,Z 53,A -2.4476,B 0,C 0,E1 0.1598,E2 90.0723} C_DIS
LIN {X 0.4347,Y 4.7894,Z 53,A -2.4239,B 0,C 0,E1 0.1598,E2 90.0723} C_DIS
LIN {X 1.0853,Y 4.6854,Z 53,A -2.4044,B 0,C 0,E1 0.1598,E2 90.0723} C_DIS
LIN {X 1.7154,Y 4.4932,Z 53,A -2.3893,B 0,C 0,E1 0.1598,E2 90.0723} C_DIS
LIN {X 2.3134,Y 4.2165,Z 53,A -2.379,B 0,C 0,E1 0.1598,E2 90.0723} C_DIS
LIN {X 2.8665,Y 3.8586,Z 53,A -2.3738,B 0,C 0,E1 0.1598,E2 90.0723} C_DIS
LIN {X 3.3672,Y 3.4308,Z 53,A -2.3736,B 0,C 0,E1 0.1598,E2 90.0723} C_DIS
LIN {X 3.805,Y 2.9388,Z 53,A -2.3784,B 0,C 0,E1 0.1598,E2 90.0723} C_DIS
LIN {X 4.1712,Y 2.3913,Z 53,A -2.3882,B 0,C 0,E1 0.1598,E2 90.0723} C_DIS
LIN {X 4.4594,Y 1.799,Z 53,A -2.4028,B 0,C 0,E1 0.1598,E2 90.0722} C_DIS
LIN {X 4.6646,Y 1.1729,Z 53,A -2.422,B 0,C 0,E1 0.1598,E2 90.0722} C_DIS
LIN {X 4.7809,Y 0.5244,Z 53,A -2.4453,B 0,C 0,E1 0.1598,E2 90.0721} C_DIS
LIN {X 4.8072,Y -0.1338,Z 53,A -2.4724,B 0,C 0,E1 0.1598,E2 90.0721} C_DIS
LIN {X 4.7431,Y -0.7894,Z 53,A -2.5028,B 0,C 0,E1 0.1598,E2 90.072} C_DIS
LIN {X 4.5908,Y -1.4303,Z 53,A -2.5357,B 0,C 0,E1 0.1598,E2 90.072} C_DIS
LIN {X 4.3507,Y -2.0437,Z 53,A -2.5708,B 0,C 0,E1 0.1598,E2 90.072} C_DIS
LIN {X 4.0313,Y -2.6197,Z 53,A -2.6071,B 0,C 0,E1 0.1598,E2 90.072} C_DIS
LIN {X 3.6341,Y -3.1451,Z 53,A -2.6442,B 0,C 0,E1 0.1598,E2 90.072} C_DIS
LIN {X 3.1722,Y -3.6146,Z 53,A -2.6812,B 0,C 0,E1 0.1598,E2 90.0719} C_DIS
LIN {X 2.6481,Y -4.0134,Z 53,A -2.7175,B 0,C 0,E1 0.1598,E2 90.0719} C_DIS
LIN {X 2.0742,Y -4.3369,Z 53,A -2.7524,B 0,C 0,E1 0.1598,E2 90.0719} C_DIS
LIN {X 1.462,Y -4.5798,Z 53,A -2.7852,B 0,C 0,E1 0.1598,E2 90.0719} C_DIS
LIN {X 0.8224,Y -4.7376,Z 53,A -2.8154,B 0,C 0,E1 0.1598,E2 90.0719} C_DIS
LIN {X 0.0024,Y -4.8127,Z 53,A -2.8487,B 0,C 0,E1 0.1598,E2 90.0718} C_DIS
Enddeposition()
LIN {X 0.0024,Y -4.8127,Z 53,A -2.8487,B 0,C 0,E1 0.1598,E2 90.0718} C_DIS
Startdeposition()
$VEL.CP = VEL_PRINT
LIN {X 0.2255,Y -5.7065,Z 53,A -88.058,B 6.4325,C -0.2436,E1 6.4504,E2 174.4545} C_DIS
LIN {X 1.0436,Y -5.6174,Z 53,A -79.6089,B 6.4323,C -0.2482,E1 6.4737,E2 166.0002} C_DIS
LIN {X 1.84,Y -5.4088,Z 53,A -71.3643,B 6.432,C -0.2558,E1 6.4958,E2 157.7511} C_DIS
LIN {X 2.5975,Y -5.087,Z 53,A -63.3868,B 6.4316,C -0.266,E1 6.516,E2 149.77} C_DIS
LIN {X 3.3026,Y -4.6626,Z 53,A -55.1183,B 6.431,C -0.2795,E1 6.5353,E2 141.4964} C_DIS
LIN {X 3.9376,Y -4.1388,Z 53,A -46.8352,B 6.4303,C -0.2957,E1 6.5526,E2 133.2079} C_DIS
LIN {X 4.4915,Y -3.53,Z 53,A -39.0387,B 6.4295,C -0.3127,E1 6.5666,E2 125.4086} C_DIS
LIN {X 4.9534,Y -2.8487,Z 53,A -32.9324,B 6.4288,C -0.3263,E1 6.5759,E2 119.308} C_DIS
LIN {X 5.347,Y -2.0255,Z 53,A -21.3288,B 6.4272,C -0.3577,E1 6.5891,E2 107.6872} C_DIS
LIN {X 5.6362,Y -0.9251,Z 53,A -10.6518,B 6.4255,C -0.3869,E1 6.5956,E2 97.0076} C_DIS
LIN {X 5.7102,Y -0.1171,Z 53,A -2.7563,B 6.4241,C -0.409,E1 6.5969,E2 89.1097} C_DIS
LIN {X 5.6681,Y 0.6932,Z 53,A 5.1855,B 6.4227,C -0.4311,E1 6.5949,E2 81.1656} C_DIS
LIN {X 5.5132,Y 1.4895,Z 53,A 13.018,B 6.4212,C -0.4524,E1 6.59,E2 73.3321} C_DIS
LIN {X 5.2469,Y 2.2559,Z 53,A 21.0193,B 6.4197,C -0.4732,E1 6.5819,E2 65.3296} C_DIS
LIN {X 4.8744,Y 2.9768,Z 53,A 29.0778,B 6.4183,C -0.4929,E1 6.5709,E2 57.2702} C_DIS
LIN {X 4.4035,Y 3.6377,Z 53,A 36.883,B 6.4169,C -0.5101,E1 6.5576,E2 49.4661} C_DIS
LIN {X 3.8442,Y 4.2256,Z 53,A 45.2676,B 6.4156,C -0.5266,E1 6.5409,E2 41.0807} C_DIS
LIN {X 3.2057,Y 4.7265,Z 53,A 53.004,B 6.4146,C -0.5392,E1 6.5234,E2 33.347} C_DIS
LIN {X 2.5036,Y 5.1332,Z 53,A 61.1532,B 6.4136,C -0.5501,E1 6.5034,E2 25.1994} C_DIS
LIN {X 1.7508,Y 5.4358,Z 53,A 69.1801,B 6.413,C -0.5578,E1 6.4823,E2 17.1751} C_DIS
LIN {X 0.9631,Y 5.6315,Z 53,A 77.2112,B 6.4126,C -0.5625,E1 6.4604,E2 9.1475} C_DIS
LIN {X 0.1554,Y 5.71,Z 53,A 85.6176,B 6.4124,C -0.5642,E1 6.437,E2 0.7435} C_DIS
LIN {X -0.6553,Y 5.6735,Z 53,A 93.6908,B 6.4126,C -0.5624,E1 6.4145,E2 -7.3255} C_DIS
LIN {X -1.4523,Y 5.5216,Z 53,A 101.6254,B 6.413,C -0.5576,E1 6.3929,E2 -15.255} C_DIS
LIN {X -2.2208,Y 5.2618,Z 53,A 110.0999,B 6.4137,C -0.5494,E1 6.3708,E2 -23.726} C_DIS
LIN {X -2.9439,Y 4.8936,Z 53,A 118.2249,B 6.4146,C -0.5384,E1 6.351,E2 -31.8461} C_DIS
LIN {X -3.6073,Y 4.4266,Z 53,A 126.5707,B 6.4158,C -0.5244,E1 6.3325,E2 -40.1876} C_DIS
LIN {X -4.1993,Y 3.8716,Z 53,A 134.6383,B 6.4171,C -0.5082,E1 6.3166,E2 -48.2499} C_DIS
LIN {X -4.7057,Y 3.2376,Z 53,A 143.3547,B 6.4186,C -0.4888,E1 6.3021,E2 -56.9634} C_DIS
LIN {X -5.1156,Y 2.5372,Z 53,A 151.4778,B 6.4201,C -0.4686,E1 6.2914,E2 -65.0818} C_DIS
LIN {X -5.4236,Y 1.7867,Z 53,A 159.7812,B 6.4216,C -0.4467,E1 6.2834,E2 -73.3813} C_DIS
LIN {X -5.6225,Y 1.0001,Z 53,A 168.0177,B 6.4232,C -0.424,E1 6.2785,E2 -81.6139} C_DIS
LIN {X -5.7085,Y 0.1934,Z 53,A 176.4524,B 6.4247,C -0.4005,E1 6.2769,E2 -90.0461} C_DIS
LIN {X -5.6795,Y -0.6175,Z 53,A -175.0863,B 6.4261,C -0.3769,E1 6.2786,E2 -98.5054} C_DIS
LIN {X -5.5356,Y -1.4164,Z 53,A -169.1127,B 6.4271,C -0.3594,E1 6.2818,E2 -104.4676} C_DIS
LIN {X -5.2978,Y -2.1489,Z 53,A -157.3284,B 6.4286,C -0.3305,E1 6.293,E2 -116.2667} C_DIS
LIN {X -4.9317,Y -2.8955,Z 53,A -148.2121,B 6.4297,C -0.3091,E1 6.3058,E2 -125.3853} C_DIS
LIN {X -4.1264,Y -3.9574,Z 53,A -136.266,B 6.4309,C -0.2835,E1 6.3273,E2 -137.3247} C_DIS
LIN {X -3.3103,Y -4.6621,Z 53,A -126.7995,B 6.4316,C -0.2668,E1 6.3478,E2 -146.786} C_DIS
LIN {X -2.6573,Y -5.0636,Z 53,A -117.7746,B 6.432,C -0.2557,E1 6.3697,E2 -155.8185} C_DIS
LIN {X -1.7394,Y -5.4404,Z 53,A -107.7231,B 6.4324,C -0.2469,E1 6.396,E2 -165.8736} C_DIS
LIN {X -0.9683,Y -5.6279,Z 53,A -99.9561,B 6.4325,C -0.2433,E1 6.4172,E2 -173.6426} C_DIS
LIN {X 0.0196,Y -5.7138,Z 53,A -94.0315,B 6.4326,C -0.2407,E1 6.4336,E2 -179.5521} C_DIS
Enddeposition()
LIN {X 0.0196,Y -5.7138,Z 53,A -94.0315,B 6.4326,C -0.2407,E1 6.4336,E2 -179.5521} C_DIS
Startdeposition()
$VEL.CP = VEL_PRINT
LIN {X -0.4921,Y -6.6008,Z 53,A -99.7047,B 12.3354,C -0.8665,E1 12.3504,E2 -175.0912} C_DIS
LIN {X -1.1795,Y -6.514,Z 53,A -105.7992,B 12.3353,C -0.8682,E1 12.3336,E2 -168.994} C_DIS
LIN {X -1.854,Y -6.3548,Z 53,A -111.8138,B 12.335,C -0.8718,E1 12.3174,E2 -162.9777} C_DIS
LIN {X -2.5085,Y -6.1268,Z 53,A -117.7545,B 12.3347,C -0.8772,E1 12.3018,E2 -157.0361} C_DIS
LIN {X -3.1356,Y -5.832,Z 53,A -123.8724,B 12.3342,C -0.8842,E1 12.2866,E2 -150.917} C_DIS
LIN {X -3.7281,Y -5.4725,Z 53,A -129.923,B 12.3336,C -0.8929,E1 12.2724,E2 -144.866} C_DIS
LIN {X -4.2798,Y -5.0531,Z 53,A -136.0682,B 12.3328,C -0.9032,E1 12.259,E2 -138.7206} C_DIS
LIN {X -4.7834,Y -4.577,Z 53,A -141.9275,B 12.332,C -0.9146,E1 12.2474,E2 -132.8631} C_DIS
LIN {X -5.2371,Y -4.0531,Z 53,A -148.0681,B 12.331,C -0.9276,E1 12.2365,E2 -126.7233} C_DIS
LIN {X -5.6302,Y -3.4824,Z 53,A -154.307,B 12.33,C -0.942,E1 12.227,E2 -120.4855} C_DIS
LIN {X -5.9628,Y -2.8744,Z 53,A -160.4765,B 12.3288,C -0.9573,E1 12.2191,E2 -114.3178} C_DIS
LIN {X -6.2293,Y -2.2347,Z 53,A -166.0408,B 12.3276,C -0.9724,E1 12.2135,E2 -108.7584} C_DIS
LIN {X -6.4318,Y -1.5721,Z 53,A -172.4148,B 12.3263,C -0.9894,E1 12.2088,E2 -102.3861} C_DIS
LIN {X -6.5607,Y -0.8912,Z 53,A -178.4277,B 12.325,C -1.0064,E1 12.2061,E2 -96.3769} C_DIS
LIN {X -6.6188,Y -0.2007,Z 53,A 175.4651,B 12.3236,C -1.0237,E1 12.2051,E2 -90.2734} C_DIS
LIN {X -6.6022,Y 0.492,Z 53,A 169.3272,B 12.3221,C -1.0412,E1 12.2059,E2 -84.1394} C_DIS
LIN {X -6.5151,Y 1.1795,Z 53,A 163.2718,B 12.3207,C -1.0584,E1 12.2085,E2 -78.0884} C_DIS
LIN {X -6.356,Y 1.8539,Z 53,A 157.2293,B 12.3192,C -1.0752,E1 12.2128,E2 -72.0506} C_DIS
LIN {X -6.1276,Y 2.5082,Z 53,A 151.1604,B 12.3178,C -1.0916,E1 12.2188,E2 -65.9865} C_DIS
LIN {X -5.8322,Y 3.1351,Z 53,A 144.8967,B 12.3164,C -1.1076,E1 12.2267,E2 -59.7268} C_DIS
LIN {X -5.4706,Y 3.7263,Z 53,A 139.1856,B 12.3151,C -1.122,E1 12.2353,E2 -54.022} C_DIS
LIN {X -5.0525,Y 4.279,Z 53,A 132.658,B 12.3138,C -1.1363,E1 12.2467,E2 -47.4974} C_DIS
LIN {X -4.5763,Y 4.7826,Z 53,A 126.832,B 12.3127,C -1.1486,E1 12.2582,E2 -41.6771} C_DIS
LIN {X -4.0518,Y 5.2355,Z 53,A 121.1751,B 12.3117,C -1.1596,E1 12.2703,E2 -36.0265} C_DIS
LIN {X -3.4835,Y 5.6321,Z 53,A 114.7314,B 12.3108,C -1.1697,E1 12.2854,E2 -29.5857} C_DIS
LIN {X -2.8756,Y 5.9649,Z 53,A 108.6843,B 12.31,C -1.1779,E1 12.3004,E2 -23.5428} C_DIS
LIN {X -2.2362,Y 6.2323,Z 53,A 102.5231,B 12.3094,C -1.1845,E1 12.3164,E2 -17.3851} C_DIS
LIN {X -1.5719,Y 6.4296,Z 53,A 96.7909,B 12.3089,C -1.1895,E1 12.3318,E2 -11.658} C_DIS
LIN {X -0.8915,Y 6.5605,Z 53,A 90.6434,B 12.3086,C -1.1925,E1 12.3487,E2 -5.5133} C_DIS
LIN {X -0.2008,Y 6.6161,Z 53,A 84.4181,B 12.3085,C -1.1937,E1 12.3661,E2 0.7099} C_DIS
LIN {X 0.492,Y 6.6011,Z 53,A 78.7741,B 12.3085,C -1.1937,E1 12.3818,E2 6.3498} C_DIS
LIN {X 1.1794,Y 6.513,Z 53,A 72.5633,B 12.3087,C -1.1911,E1 12.3989,E2 12.5595} C_DIS
LIN {X 1.8535,Y 6.3534,Z 53,A 66.8513,B 12.3091,C -1.1876,E1 12.4144,E2 18.2685} C_DIS
LIN {X 2.5083,Y 6.1264,Z 53,A 60.8323,B 12.3096,C -1.1819,E1 12.4301,E2 24.2866} C_DIS
LIN {X 3.1356,Y 5.832,Z 53,A 54.5529,B 12.3104,C -1.1738,E1 12.4457,E2 30.5667} C_DIS
LIN {X 3.7264,Y 5.47,Z 53,A 48.7117,B 12.3112,C -1.1653,E1 12.4594,E2 36.4071} C_DIS
LIN {X 4.2776,Y 5.05,Z 53,A 43.0101,B 12.3121,C -1.1557,E1 12.4718,E2 42.1078} C_DIS
LIN {X 4.784,Y 4.5769,Z 53,A 37.0376,B 12.3131,C -1.144,E1 12.4837,E2 48.0813} C_DIS
LIN {X 5.2374,Y 4.0527,Z 53,A 30.9726,B 12.3143,C -1.1307,E1 12.4945,E2 54.1482} C_DIS
LIN {X 5.6326,Y 3.4833,Z 53,A 24.9913,B 12.3156,C -1.1167,E1 12.5036,E2 60.1315} C_DIS
LIN {X 5.9636,Y 2.8745,Z 53,A 18.7317,B 12.317,C -1.1007,E1 12.5116,E2 66.395} C_DIS
LIN {X 6.2295,Y 2.2345,Z 53,A 13.1982,B 12.3183,C -1.0865,E1 12.5171,E2 71.9289} C_DIS
LIN {X 6.4303,Y 1.5713,Z 53,A 7.3228,B 12.3196,C -1.0705,E1 12.5215,E2 77.8072} C_DIS
LIN {X 6.5596,Y 0.8905,Z 53,A 1.2019,B 12.3211,C -1.0531,E1 12.5242,E2 83.9326} C_DIS
LIN {X 6.6151,Y 0.1998,Z 53,A -4.5037,B 12.3224,C -1.0371,E1 12.5251,E2 89.6407} C_DIS
LIN {X 6.6021,Y -0.493,Z 53,A -10.4378,B 12.3238,C -1.0201,E1 12.5244,E2 95.579} C_DIS
LIN {X 6.5149,Y -1.1804,Z 53,A -16.4747,B 12.3252,C -1.0028,E1 12.5218,E2 101.6208} C_DIS
LIN {X 6.3558,Y -1.8548,Z 53,A -22.3615,B 12.3265,C -0.9864,E1 12.5176,E2 107.5119} C_DIS
LIN {X 6.1273,Y -2.509,Z 53,A -28.2826,B 12.3278,C -0.9703,E1 12.5118,E2 113.4376} C_DIS
LIN {X 5.8318,Y -3.1358,Z 53,A -34.2037,B 12.329,C -0.9549,E1 12.5043,E2 119.3635} C_DIS
LIN {X 5.4723,Y -3.7283,Z 53,A -40.4207,B 12.3302,C -0.9392,E1 12.4949,E2 125.5869} C_DIS
LIN {X 5.0513,Y -4.2789,Z 53,A -45.8005,B 12.3311,C -0.9274,E1 12.4855,E2 130.9683} C_DIS
LIN {X 4.5779,Y -4.7849,Z 53,A -52.0224,B 12.332,C -0.9139,E1 12.4733,E2 137.1967} C_DIS
LIN {X 4.052,Y -5.2362,Z 53,A -57.9736,B 12.3329,C -0.9025,E1 12.4604,E2 143.1525} C_DIS
LIN {X 3.4832,Y -5.6323,Z 53,A -63.9724,B 12.3336,C -0.8924,E1 12.4464,E2 149.1561} C_DIS
LIN {X 2.8753,Y -5.9652,Z 53,A -69.9077,B 12.3342,C -0.8839,E1 12.4317,E2 155.0955} C_DIS
LIN {X 2.236,Y -6.2327,Z 53,A -75.9123,B 12.3347,C -0.8769,E1 12.416,E2 161.1044} C_DIS
LIN {X 1.5722,Y -6.4316,Z 53,A -81.8742,B 12.3351,C -0.8717,E1 12.4,E2 167.07} C_DIS
LIN {X 0.8912,Y -6.56,Z 53,A -87.7692,B 12.3353,C -0.8683,E1 12.3837,E2 172.9679} C_DIS
LIN {X 0.0274,Y -6.6207,Z 53,A -92.8089,B 12.3353,C -0.8692,E1 12.3697,E2 177.9981} C_DIS
Enddeposition()
LIN {X 0.0274,Y -6.6207,Z 53,A -92.8089,B 12.3353,C -0.8692,E1 12.3697,E2 177.9981} C_DIS
Startdeposition()
$VEL.CP = VEL_PRINT
LIN {X 0.069,Y -7.5291,Z 53,A -92.1649,B 18.2719,C -1.7832,E1 18.366,E2 175.9937} C_DIS
LIN {X 1.4495,Y -7.3884,Z 53,A -82.9904,B 18.2716,C -1.7861,E1 18.3914,E2 166.8216} C_DIS
LIN {X 2.3678,Y -7.1412,Z 53,A -76.0361,B 18.271,C -1.7925,E1 18.41,E2 159.8635} C_DIS
LIN {X 3.2515,Y -6.7901,Z 53,A -68.1199,B 18.2699,C -1.8044,E1 18.4303,E2 151.9367} C_DIS
LIN {X 4.2491,Y -6.209,Z 53,A -60.1997,B 18.2688,C -1.8163,E1 18.4491,E2 144.0138} C_DIS
LIN {X 5.4544,Y -5.1889,Z 53,A -46.1188,B 18.2655,C -1.85,E1 18.478,E2 129.9062} C_DIS
LIN {X 6.3786,Y -3.9949,Z 53,A -38.1973,B 18.2642,C -1.8632,E1 18.491,E2 121.9967} C_DIS
LIN {X 6.7554,Y -3.3229,Z 53,A -30.9985,B 18.2621,C -1.8848,E1 18.5007,E2 114.7821} C_DIS
LIN {X 7.0765,Y -2.5692,Z 53,A -23.4778,B 18.2597,C -1.9084,E1 18.5083,E2 107.2453} C_DIS
LIN {X 7.4367,Y -1.1733,Z 53,A -13.2878,B 18.2568,C -1.9367,E1 18.5143,E2 97.0487} C_DIS
LIN {X 7.5255,Y -0.0456,Z 53,A -6.496,B 18.2551,C -1.9536,E1 18.5155,E2 90.2599} C_DIS
LIN {X 7.496,Y 0.7141,Z 53,A 1.0792,B 18.2524,C -1.9791,E1 18.5142,E2 82.6671} C_DIS
LIN {X 7.2933,Y 1.8528,Z 53,A 9.7108,B 18.2498,C -2.0035,E1 18.5093,E2 74.0285} C_DIS
LIN {X 7.0103,Y 2.7337,Z 53,A 14.8178,B 18.2487,C -2.0141,E1 18.5048,E2 68.9283} C_DIS
LIN {X 6.6945,Y 3.4482,Z 53,A 22.3426,B 18.2463,C -2.0366,E1 18.4958,E2 61.3893} C_DIS
LIN {X 6.0843,Y 4.4371,Z 53,A 31.5645,B 18.2438,C -2.0593,E1 18.4816,E2 52.1597} C_DIS
LIN {X 5.4709,Y 5.1648,Z 53,A 38.1961,B 18.2424,C -2.0724,E1 18.4694,E2 45.5283} C_DIS
LIN {X 4.9212,Y 5.6914,Z 53,A 43.9348,B 18.2412,C -2.0831,E1 18.4575,E2 39.788} C_DIS
LIN {X 4.1667,Y 6.2715,Z 53,A 51.9353,B 18.2397,C -2.0972,E1 18.4393,E2 31.7818} C_DIS
LIN {X 3.1729,Y 6.8283,Z 53,A 60.3626,B 18.2386,C -2.1072,E1 18.4184,E2 23.3556} C_DIS
LIN {X 2.0786,Y 7.2379,Z 53,A 69.3949,B 18.2377,C -2.1147,E1 18.3945,E2 14.3237} C_DIS
LIN {X 1.1421,Y 7.4417,Z 53,A 76.4953,B 18.2374,C -2.1173,E1 18.375,E2 7.2265} C_DIS
LIN {X 0.1239,Y 7.5279,Z 53,A 84.31,B 18.2374,C -2.1175,E1 18.3532,E2 -0.5851} C_DIS
LIN {X -0.9889,Y 7.4648,Z 53,A 92.631,B 18.2378,C -2.1139,E1 18.3301,E2 -8.9004} C_DIS
LIN {X -2.3382,Y 7.1568,Z 53,A 103.8326,B 18.2388,C -2.1051,E1 18.3,E2 -20.0976} C_DIS
LIN {X -3.4632,Y 6.68,Z 53,A 112.257,B 18.2402,C -2.0922,E1 18.2787,E2 -28.5097} C_DIS
LIN {X -4.1505,Y 6.2762,Z 53,A 118.3287,B 18.2413,C -2.0821,E1 18.2643,E2 -34.5757} C_DIS
LIN {X -4.7917,Y 5.8029,Z 53,A 124.5853,B 18.2426,C -2.0703,E1 18.2506,E2 -40.827} C_DIS
LIN {X -5.3777,Y 5.2626,Z 53,A 130.4444,B 18.2441,C -2.0574,E1 18.2388,E2 -46.6788} C_DIS
LIN {X -6.1277,Y 4.3748,Z 53,A 138.874,B 18.2463,C -2.0364,E1 18.2241,E2 -55.0964} C_DIS
LIN {X -6.5647,Y 3.6857,Z 53,A 145.363,B 18.2481,C -2.0201,E1 18.2147,E2 -61.5797} C_DIS
LIN {X -6.9641,Y 2.8612,Z 53,A 153.3744,B 18.2502,C -1.9999,E1 18.2055,E2 -69.588} C_DIS
LIN {X -7.257,Y 2.0045,Z 53,A 160.2802,B 18.2523,C -1.9801,E1 18.1999,E2 -76.4861} C_DIS
LIN {X -7.4736,Y 0.8803,Z 53,A 168.4934,B 18.2549,C -1.9551,E1 18.1962,E2 -84.6876} C_DIS
LIN {X -7.5251,Y 0.0651,Z 53,A 174.8988,B 18.2568,C -1.9365,E1 18.1956,E2 -91.0873} C_DIS
LIN {X -7.4517,Y -1.0802,Z 53,A -175.8759,B 18.2595,C -1.9103,E1 18.1981,E2 -100.3063} C_DIS
LIN {X -7.2578,Y -2.0038,Z 53,A -168.6407,B 18.2615,C -1.8899,E1 18.2029,E2 -107.5354} C_DIS
LIN {X -6.8577,Y -3.0977,Z 53,A -159.9862,B 18.2639,C -1.8663,E1 18.2118,E2 -116.1821} C_DIS
LIN {X -6.3392,Y -4.0626,Z 53,A -150.8906,B 18.266,C -1.8452,E1 18.2247,E2 -125.2761} C_DIS
LIN {X -5.6635,Y -4.9546,Z 53,A -143.2358,B 18.2677,C -1.8269,E1 18.2381,E2 -132.9221} C_DIS
LIN {X -5.174,Y -5.4648,Z 53,A -137.7705,B 18.2688,C -1.8163,E1 18.2489,E2 -138.3858} C_DIS
LIN {X -4.6375,Y -5.9251,Z 53,A -132.5156,B 18.2697,C -1.8069,E1 18.2602,E2 -143.6385} C_DIS
LIN {X -3.9132,Y -6.4315,Z 53,A -125.2917,B 18.2706,C -1.7971,E1 18.2771,E2 -150.864} C_DIS
LIN {X -3.2321,Y -6.7995,Z 53,A -119.2732,B 18.2712,C -1.7903,E1 18.2922,E2 -156.8831} C_DIS
LIN {X -2.1176,Y -7.2202,Z 53,A -110.3637,B 18.2719,C -1.7828,E1 18.3156,E2 -165.7929} C_DIS
LIN {X -0.9257,Y -7.4719,Z 53,A -100.9189,B 18.2722,C -1.7799,E1 18.3416,E2 -175.2413} C_DIS
LIN {X 0.0028,Y -7.5273,Z 53,A -97.21,B 18.2728,C -1.7739,E1 18.3519,E2 -178.9326} C_DIS
Enddeposition()
LIN {X 0.0028,Y -7.5273,Z 53,A -97.21,B 18.2728,C -1.7739,E1 18.3519,E2 -178.9326} C_DIS
Startdeposition()
$VEL.CP = VEL_PRINT
LIN {X -0.0818,Y -8.4342,Z 53,A -100.3163,B 24.1651,C -2.9888,E1 24.33,E2 -177.325} C_DIS
LIN {X -1.5271,Y -8.2913,Z 53,A -109.3001,B 24.1646,C -2.9928,E1 24.3052,E2 -168.3442} C_DIS
LIN {X -2.2196,Y -8.1372,Z 53,A -114.5165,B 24.1644,C -2.9947,E1 24.2911,E2 -163.1244} C_DIS
LIN {X -3.3876,Y -7.7195,Z 53,A -122.5681,B 24.1634,C -3.0031,E1 24.2702,E2 -155.0756} C_DIS
LIN {X -4.1601,Y -7.3307,Z 53,A -128.2772,B 24.1625,C -3.0107,E1 24.2561,E2 -149.3688} C_DIS
LIN {X -5.0672,Y -6.7425,Z 53,A -136.6353,B 24.1613,C -3.0213,E1 24.237,E2 -141.0072} C_DIS
LIN {X -6.112,Y -5.8112,Z 53,A -145.8108,B 24.159,C -3.0404,E1 24.2186,E2 -131.8392} C_DIS
LIN {X -6.9176,Y -4.8245,Z 53,A -153.9489,B 24.1566,C -3.0605,E1 24.2047,E2 -123.7106} C_DIS
LIN {X -7.4437,Y -3.9588,Z 53,A -160.7007,B 24.1545,C -3.0782,E1 24.1953,E2 -116.966} C_DIS
LIN {X -7.9044,Y -2.9413,Z 53,A -168.6327,B 24.152,C -3.0991,E1 24.1867,E2 -109.0402} C_DIS
LIN {X -8.2123,Y -1.9051,Z 53,A -176.0404,B 24.1494,C -3.1206,E1 24.1813,E2 -101.641} C_DIS
LIN {X -8.393,Y -0.8392,Z 53,A 176.3878,B 24.1467,C -3.1428,E1 24.1784,E2 -94.0773} C_DIS
LIN {X -8.4276,Y 0.373,Z 53,A 167.5398,B 24.1435,C -3.1685,E1 24.1785,E2 -85.2375} C_DIS
LIN {X -8.2793,Y 1.6128,Z 53,A 158.539,B 24.1403,C -3.1948,E1 24.1825,E2 -76.2464} C_DIS
LIN {X -7.9188,Y 2.9022,Z 53,A 150.4718,B 24.1369,C -3.2216,E1 24.1894,E2 -68.1973} C_DIS
LIN {X -7.528,Y 3.8043,Z 53,A 143.9247,B 24.1345,C -3.2407,E1 24.197,E2 -61.6604} C_DIS
LIN {X -7.0456,Y 4.6391,Z 53,A 136.6451,B 24.1323,C -3.2586,E1 24.2077,E2 -54.3865} C_DIS
LIN {X -6.3121,Y 5.5886,Z 53,A 129.049,B 24.1296,C -3.2791,E1 24.2211,E2 -46.8044} C_DIS
LIN {X -5.7089,Y 6.2032,Z 53,A 123.1442,B 24.1279,C -3.2924,E1 24.2329,E2 -40.9069} C_DIS
LIN {X -5.0466,Y 6.7537,Z 53,A 117.1617,B 24.1264,C -3.3044,E1 24.246,E2 -34.931} C_DIS
LIN {X -4.3302,Y 7.2314,Z 53,A 111.5313,B 24.125,C -3.3151,E1 24.2593,E2 -29.3085} C_DIS
LIN {X -3.2715,Y 7.7735,Z 53,A 103.6281,B 24.1234,C -3.3274,E1 24.2791,E2 -21.4144} C_DIS
LIN {X -2.3543,Y 8.1003,Z 53,A 95.9753,B 24.1226,C -3.3333,E1 24.2995,E2 -13.7619} C_DIS
LIN {X -1.1997,Y 8.3494,Z 53,A 87.956,B 24.1219,C -3.3391,E1 24.3215,E2 -5.7485} C_DIS
LIN {X -0.071,Y 8.4348,Z 53,A 80.3298,B 24.1216,C -3.3416,E1 24.3427,E2 1.8732} C_DIS
LIN {X 0.9801,Y 8.377,Z 53,A 73.5445,B 24.1216,C -3.342,E1 24.3616,E2 8.6536} C_DIS
LIN {X 2.062,Y 8.1783,Z 53,A 66.1163,B 24.1219,C -3.3388,E1 24.3818,E2 16.08} C_DIS
LIN {X 2.9946,Y 7.8848,Z 53,A 59.7368,B 24.1225,C -3.3342,E1 24.3987,E2 22.4577} C_DIS
LIN {X 3.8518,Y 7.4998,Z 53,A 53.5507,B 24.1234,C -3.3277,E1 24.4143,E2 28.6432} C_DIS
LIN {X 4.8058,Y 6.9305,Z 53,A 45.6143,B 24.125,C -3.3149,E1 24.433,E2 36.5846} C_DIS
LIN {X 5.8834,Y 6.0434,Z 53,A 35.9012,B 24.1275,C -3.296,E1 24.4534,E2 46.3042} C_DIS
LIN {X 6.6314,Y 5.2113,Z 53,A 28.6699,B 24.1294,C -3.2809,E1 24.4665,E2 53.5383} C_DIS
LIN {X 7.2653,Y 4.2864,Z 53,A 20.0112,B 24.1325,C -3.2566,E1 24.4794,E2 62.2111} C_DIS
LIN {X 7.9588,Y 2.7934,Z 53,A 9.5017,B 24.136,C -3.2293,E1 24.4907,E2 72.7276} C_DIS
LIN {X 8.2902,Y 1.5314,Z 53,A 2.7094,B 24.1378,C -3.2148,E1 24.4953,E2 79.5147} C_DIS
LIN {X 8.4002,Y 0.774,Z 53,A -4.487,B 24.1412,C -3.1876,E1 24.4977,E2 86.7333} C_DIS
LIN {X 8.4293,Y -0.312,Z 53,A -11.1161,B 24.1435,C -3.1691,E1 24.4977,E2 93.3667} C_DIS
LIN {X 8.3448,Y -1.2283,Z 53,A -16.8618,B 24.1455,C -3.1527,E1 24.4959,E2 99.1173} C_DIS
LIN {X 8.0965,Y -2.367,Z 53,A -26.052,B 24.1493,C -3.1214,E1 24.4898,E2 108.3288} C_DIS
LIN {X 7.7856,Y -3.2431,Z 53,A -32.2389,B 24.1515,C -3.1035,E1 24.4835,E2 114.5238} C_DIS
LIN {X 7.2719,Y -4.2661,Z 53,A -38.7996,B 24.1533,C -3.0882,E1 24.4749,E2 121.0861} C_DIS
LIN {X 6.5664,Y -5.2956,Z 53,A -49.0009,B 24.1571,C -3.0571,E1 24.4579,E2 131.3127} C_DIS
LIN {X 5.8204,Y -6.1033,Z 53,A -55.754,B 24.1587,C -3.0432,E1 24.4446,E2 138.0701} C_DIS
LIN {X 4.9522,Y -6.8292,Z 53,A -63.3293,B 24.1605,C -3.0278,E1 24.4279,E2 145.6541} C_DIS
LIN {X 4.1033,Y -7.3684,Z 53,A -71.0481,B 24.1624,C -3.0121,E1 24.4093,E2 153.387} C_DIS
LIN {X 2.6455,Y -8.0094,Z 53,A -80.7267,B 24.1635,C -3.0022,E1 24.3841,E2 163.0677} C_DIS
LIN {X 1.7024,Y -8.2605,Z 53,A -87.1992,B 24.1642,C -2.9966,E1 24.3665,E2 169.5444} C_DIS
LIN {X 0.6524,Y -8.4062,Z 53,A -94.3657,B 24.1646,C -2.9926,E1 24.3467,E2 176.7152} C_DIS
LIN {X 0.6524,Y -8.4062,Z 53,A -94.3657,B 24.1646,C -2.9926,E1 24.3467,E2 176.7152} C_DIS
Enddeposition()
LIN {X 0.0327,Y -9.3355,Z 53,A -96.434,B 24.8146,C -3.1404,E1 25.0031,E2 178.6233} C_DIS
Startdeposition()
$VEL.CP = VEL_PRINT
LIN {X 1.0931,Y -9.2755,Z 53,A -89.0877,B 24.8138,C -3.1465,E1 25.0236,E2 171.2665} C_DIS
LIN {X 2.2259,Y -9.0712,Z 53,A -82.4915,B 24.8133,C -3.1506,E1 25.0416,E2 164.6687} C_DIS
LIN {X 3.4047,Y -8.6986,Z 53,A -74.2199,B 24.8119,C -3.1629,E1 25.0635,E2 156.3843} C_DIS
LIN {X 4.2688,Y -8.308,Z 53,A -68.63,B 24.8109,C -3.171,E1 25.0775,E2 150.79} C_DIS
LIN {X 5.217,Y -7.7469,Z 53,A -61.9684,B 24.8095,C -3.183,E1 25.0932,E2 144.1213} C_DIS
LIN {X 6.0143,Y -7.1452,Z 53,A -55.6926,B 24.8078,C -3.1968,E1 25.1069,E2 137.8364} C_DIS
LIN {X 6.9081,Y -6.2875,Z 53,A -48.1803,B 24.8057,C -3.2143,E1 25.1216,E2 130.3147} C_DIS
LIN {X 7.5738,Y -5.4673,Z 53,A -40.914,B 24.8031,C -3.2358,E1 25.1338,E2 123.0322} C_DIS
LIN {X 8.3311,Y -4.2221,Z 53,A -33.7728,B 24.8013,C -3.2502,E1 25.1436,E2 115.8938} C_DIS
LIN {X 8.6571,Y -3.5073,Z 53,A -28.0059,B 24.7989,C -3.27,E1 25.15,E2 110.1115} C_DIS
LIN {X 9.0333,Y -2.3715,Z 53,A -20.8872,B 24.7963,C -3.2909,E1 25.1557,E2 102.9837} C_DIS
LIN {X 9.2576,Y -1.2449,Z 53,A -13.3808,B 24.7932,C -3.3156,E1 25.159,E2 95.463} C_DIS
LIN {X 9.3411,Y 0.0023,Z 53,A -6.6669,B 24.7909,C -3.3334,E1 25.1597,E2 88.7466} C_DIS
LIN {X 9.2862,Y 0.9985,Z 53,A -0.3574,B 24.7884,C -3.3534,E1 25.1584,E2 82.4271} C_DIS
LIN {X 9.1118,Y 2.0281,Z 53,A 5.625,B 24.7863,C -3.3702,E1 25.1553,E2 76.44} C_DIS
LIN {X 8.8339,Y 3.0347,Z 53,A 12.6049,B 24.7835,C -3.3921,E1 25.1495,E2 69.4478} C_DIS
LIN {X 8.4062,Y 4.069,Z 53,A 19.4565,B 24.7811,C -3.4109,E1 25.1417,E2 62.5889} C_DIS
LIN {X 7.8873,Y 5.0022,Z 53,A 26.1224,B 24.7788,C -3.4282,E1 25.1321,E2 55.9158} C_DIS
LIN {X 7.1588,Y 5.9984,Z 53,A 33.17,B 24.7769,C -3.443,E1 25.1201,E2 48.8664} C_DIS
LIN {X 6.5539,Y 6.6554,Z 53,A 38.9451,B 24.7752,C -3.4559,E1 25.1088,E2 43.0854} C_DIS
LIN {X 5.8362,Y 7.2931,Z 53,A 44.861,B 24.7738,C -3.4668,E1 25.0961,E2 37.1664} C_DIS
LIN {X 4.9192,Y 7.9359,Z 53,A 51.0346,B 24.7728,C -3.4744,E1 25.0818,E2 30.9954} C_DIS
LIN {X 4.0744,Y 8.4036,Z 53,A 57.5469,B 24.7715,C -3.4843,E1 25.0657,E2 24.4776} C_DIS
LIN {X 2.9777,Y 8.8539,Z 53,A 65.0838,B 24.7705,C -3.4918,E1 25.0459,E2 16.9387} C_DIS
LIN {X 1.7208,Y 9.176,Z 53,A 72.4931,B 24.7702,C -3.4939,E1 25.0258,E2 9.5345} C_DIS
LIN {X 0.4627,Y 9.3296,Z 53,A 80.5739,B 24.77,C -3.4955,E1 25.0034,E2 1.4547} C_DIS
LIN {X -0.6617,Y 9.3137,Z 53,A 86.7742,B 24.7705,C -3.4916,E1 24.9861,E2 -4.7373} C_DIS
LIN {X -1.8479,Y 9.1551,Z 53,A 94.6834,B 24.771,C -3.4879,E1 24.9643,E2 -12.6449} C_DIS
LIN {X -3.1177,Y 8.8043,Z 53,A 103.0067,B 24.7721,C -3.4795,E1 24.9421,E2 -20.9625} C_DIS
LIN {X -4.3514,Y 8.2652,Z 53,A 111.3642,B 24.7737,C -3.4673,E1 24.9211,E2 -29.3119} C_DIS
LIN {X -5.1107,Y 7.8193,Z 53,A 116.912,B 24.775,C -3.4576,E1 24.908,E2 -34.8543} C_DIS
LIN {X -6.1141,Y 7.0574,Z 53,A 122.4939,B 24.7773,C -3.4397,E1 24.8958,E2 -40.4139} C_DIS
LIN {X -6.6699,Y 6.5387,Z 53,A 129.1581,B 24.7785,C -3.4304,E1 24.8824,E2 -47.0836} C_DIS
LIN {X -7.4484,Y 5.6303,Z 53,A 134.4757,B 24.781,C -3.4111,E1 24.8729,E2 -52.3793} C_DIS
LIN {X -7.893,Y 4.993,Z 53,A 141.1235,B 24.7826,C -3.399,E1 24.8625,E2 -59.031} C_DIS
LIN {X -8.3542,Y 4.1761,Z 53,A 147.0133,B 24.7847,C -3.3827,E1 24.8548,E2 -64.9131} C_DIS
LIN {X -8.7406,Y 3.291,Z 53,A 152.9924,B 24.7869,C -3.3653,E1 24.8485,E2 -70.8837} C_DIS
LIN {X -9.1666,Y 1.7928,Z 53,A 163.7411,B 24.7906,C -3.3362,E1 24.8415,E2 -81.6254} C_DIS
LIN {X -9.3355,Y 0.2934,Z 53,A 171.8313,B 24.7942,C -3.3075,E1 24.8398,E2 -89.6954} C_DIS
LIN {X -9.3176,Y -0.6412,Z 53,A 177.6615,B 24.7964,C -3.2898,E1 24.8405,E2 -95.5182} C_DIS
LIN {X -9.1661,Y -1.7954,Z 53,A -175.1742,B 24.7991,C -3.2682,E1 24.8436,E2 -102.6733} C_DIS
LIN {X -8.8728,Y -2.904,Z 53,A -168.0958,B 24.8016,C -3.2478,E1 24.8491,E2 -109.7437} C_DIS
LIN {X -8.4536,Y -3.9714,Z 53,A -160.8916,B 24.804,C -3.2283,E1 24.857,E2 -116.9411} C_DIS
LIN {X -7.9035,Y -4.969,Z 53,A -154.296,B 24.8062,C -3.2102,E1 24.8662,E2 -123.5276} C_DIS
LIN {X -7.2968,Y -5.8311,Z 53,A -147.0744,B 24.808,C -3.1955,E1 24.8784,E2 -130.7487} C_DIS
LIN {X -6.5258,Y -6.6821,Z 53,A -139.7401,B 24.8097,C -3.1813,E1 24.8926,E2 -138.0803} C_DIS
LIN {X -5.3811,Y -7.6336,Z 53,A -130.7968,B 24.8116,C -3.1653,E1 24.9123,E2 -147.0181} C_DIS
LIN {X -4.2985,Y -8.287,Z 53,A -123.5104,B 24.8129,C -3.1541,E1 24.93,E2 -154.2992} C_DIS
LIN {X -3.5026,Y -8.6541,Z 53,A -118.2841,B 24.8136,C -3.1483,E1 24.9434,E2 -159.5239} C_DIS
LIN {X -2.3959,Y -9.027,Z 53,A -110.8521,B 24.8141,C -3.1439,E1 24.9632,E2 -166.9582} C_DIS
LIN {X -1.3601,Y -9.2365,Z 53,A -104.5912,B 24.8145,C -3.1412,E1 24.9804,E2 -173.2191} C_DIS
LIN {X -0.1491,Y -9.3387,Z 53,A -96.442,B 24.8142,C -3.1438,E1 25.0031,E2 -181.3767} C_DIS
LIN {X -0.1491,Y -9.3387,Z 53,A -96.442,B 24.8142,C -3.1438,E1 25.0031,E2 -181.3767} C_DIS
Enddeposition()
LIN {X 0.064,Y -10.2355,Z 53,A -95.7579,B 24.8161,C -3.1271,E1 25.0049,E2 -182.0208} C_DIS
Startdeposition()
$VEL.CP = VEL_PRINT
LIN {X -0.4621,Y -10.2362,Z 53,A -102.4504,B 24.8177,C -3.1136,E1 24.9862,E2 -175.2954} C_DIS
LIN {X -2.3907,Y -9.9637,Z 53,A -112.7505,B 24.8171,C -3.1189,E1 24.9579,E2 -164.9973} C_DIS
LIN {X -3.4709,Y -9.6391,Z 53,A -118.2914,B 24.8163,C -3.1255,E1 24.9432,E2 -159.4622} C_DIS
LIN {X -4.3824,Y -9.2606,Z 53,A -124.2781,B 24.8158,C -3.1303,E1 24.9279,E2 -153.4725} C_DIS
LIN {X -5.6848,Y -8.5239,Z 53,A -133.8134,B 24.8146,C -3.1402,E1 24.9053,E2 -143.9312} C_DIS
LIN {X -6.9,Y -7.5744,Z 53,A -141.3585,B 24.8125,C -3.1575,E1 24.8892,E2 -136.3983} C_DIS
LIN {X -7.6488,Y -6.8173,Z 53,A -146.8835,B 24.811,C -3.1705,E1 24.8786,E2 -130.8804} C_DIS
LIN {X -8.2939,Y -6.0171,Z 53,A -153.566,B 24.8095,C -3.183,E1 24.8673,E2 -124.196} C_DIS
LIN {X -8.9971,Y -4.8971,Z 53,A -158.8203,B 24.807,C -3.2033,E1 24.8597,E2 -118.9636} C_DIS
LIN {X -9.365,Y -4.1566,Z 53,A -164.9408,B 24.8056,C -3.2149,E1 24.8522,E2 -112.8377} C_DIS
LIN {X -9.7486,Y -3.1511,Z 53,A -171.3791,B 24.8035,C -3.2319,E1 24.8462,E2 -106.4035} C_DIS
LIN {X -10.0741,Y -1.8734,Z 53,A -178.9965,B 24.8009,C -3.2538,E1 24.8416,E2 -98.7938} C_DIS
LIN {X -10.2215,Y -0.6941,Z 53,A 174.6537,B 24.7983,C -3.2742,E1 24.8399,E2 -92.4549} C_DIS
LIN {X -10.2369,Y 0.4506,Z 53,A 168.0694,B 24.7959,C -3.294,E1 24.8402,E2 -85.8784} C_DIS
LIN {X -10.1119,Y 1.6459,Z 53,A 161.4971,B 24.7933,C -3.3148,E1 24.8425,E2 -79.3169} C_DIS
LIN {X -9.9027,Y 2.6258,Z 53,A 155.676,B 24.7911,C -3.3319,E1 24.8463,E2 -73.5027} C_DIS
LIN {X -9.5227,Y 3.7834,Z 53,A 148.4912,B 24.7886,C -3.3521,E1 24.8532,E2 -66.3256} C_DIS
LIN {X -9.0416,Y 4.8187,Z 53,A 142.4944,B 24.7862,C -3.3705,E1 24.8606,E2 -60.3406} C_DIS
LIN {X -8.5673,Y 5.6211,Z 53,A 137.1108,B 24.7844,C -3.3846,E1 24.8686,E2 -54.9635} C_DIS
LIN {X -7.9084,Y 6.5149,Z 53,A 131.2338,B 24.7824,C -3.4007,E1 24.8786,E2 -49.0973} C_DIS
LIN {X -7.1417,Y 7.3458,Z 53,A 124.4786,B 24.7805,C -3.4153,E1 24.8917,E2 -42.3479} C_DIS
LIN {X -6.381,Y 8.0164,Z 53,A 118.8055,B 24.7789,C -3.4274,E1 24.9039,E2 -36.6821} C_DIS
LIN {X -5.4701,Y 8.6626,Z 53,A 112.6096,B 24.7774,C -3.4392,E1 24.9182,E2 -30.4939} C_DIS
LIN {X -4.4101,Y 9.2451,Z 53,A 107.5887,B 24.7756,C -3.4531,E1 24.9305,E2 -25.4922} C_DIS
LIN {X -3.6456,Y 9.5749,Z 53,A 101.214,B 24.7752,C -3.4562,E1 24.947,E2 -19.1104} C_DIS
LIN {X -2.7448,Y 9.8717,Z 53,A 95.6191,B 24.7745,C -3.4613,E1 24.9619,E2 -13.5182} C_DIS
LIN {X -1.6564,Y 10.1102,Z 53,A 89.8067,B 24.7737,C -3.4671,E1 24.9778,E2 -7.7134} C_DIS
LIN {X -0.5469,Y 10.2301,Z 53,A 84.1074,B 24.7731,C -3.4716,E1 24.9936,E2 -2.0218} C_DIS
LIN {X 0.5159,Y 10.2335,Z 53,A 77.2908,B 24.7734,C -3.4697,E1 25.0127,E2 4.7983} C_DIS
LIN {X 1.556,Y 10.1264,Z 53,A 71.4506,B 24.7736,C -3.4685,E1 25.0288,E2 10.6365} C_DIS
LIN {X 2.732,Y 9.8705,Z 53,A 65.2741,B 24.7737,C -3.4671,E1 25.0456,E2 16.8077} C_DIS
LIN {X 3.9415,Y 9.4564,Z 53,A 57.2424,B 24.7751,C -3.457,E1 25.0666,E2 24.8464} C_DIS
LIN {X 5.0111,Y 8.9358,Z 53,A 50.9896,B 24.7759,C -3.4503,E1 25.0821,E2 31.0975} C_DIS
LIN {X 6.1004,Y 8.2323,Z 53,A 44.144,B 24.7772,C -3.4408,E1 25.0979,E2 37.9425} C_DIS
LIN {X 6.9122,Y 7.5636,Z 53,A 38.0473,B 24.7787,C -3.4287,E1 25.1108,E2 44.0442} C_DIS
LIN {X 7.7006,Y 6.7578,Z 53,A 31.4952,B 24.7807,C -3.4139,E1 25.1232,E2 50.6027} C_DIS
LIN {X 8.2909,Y 6.0213,Z 53,A 26.0638,B 24.7824,C -3.4006,E1 25.1323,E2 56.0397} C_DIS
LIN {X 8.8024,Y 5.2437,Z 53,A 21.1003,B 24.7839,C -3.3888,E1 25.1396,E2 61.006} C_DIS
LIN {X 9.3675,Y 4.1508,Z 53,A 14.995,B 24.7857,C -3.3749,E1 25.1471,E2 67.1117} C_DIS
LIN {X 9.7203,Y 3.2399,Z 53,A 7.9763,B 24.7889,C -3.3499,E1 25.1537,E2 74.1504} C_DIS
LIN {X 10.0601,Y 1.9437,Z 53,A 1.247,B 24.7911,C -3.3323,E1 25.1577,E2 80.8823} C_DIS
LIN {X 10.2179,Y 0.7481,Z 53,A -5.0131,B 24.7933,C -3.3147,E1 25.1596,E2 87.1471} C_DIS
LIN {X 10.2433,Y -0.1977,Z 53,A -10.6232,B 24.7956,C -3.2963,E1 25.1596,E2 92.7675} C_DIS
LIN {X 10.1213,Y -1.5873,Z 53,A -18.1924,B 24.7984,C -3.2735,E1 25.1572,E2 100.3459} C_DIS
LIN {X 9.8336,Y -2.8782,Z 53,A -25.4305,B 24.8011,C -3.2519,E1 25.1522,E2 107.5936} C_DIS
LIN {X 9.4721,Y -3.9046,Z 53,A -31.2791,B 24.8031,C -3.2352,E1 25.1465,E2 113.449} C_DIS
LIN {X 9.0436,Y -4.815,Z 53,A -37.1292,B 24.8053,C -3.2177,E1 25.1392,E2 119.3095} C_DIS
LIN {X 8.5484,Y -5.6495,Z 53,A -42.6168,B 24.8071,C -3.2024,E1 25.131,E2 124.8057} C_DIS
LIN {X 7.8901,Y -6.5363,Z 53,A -48.3538,B 24.8087,C -3.189,E1 25.1212,E2 130.5473} C_DIS
LIN {X 7.2946,Y -7.1955,Z 53,A -53.605,B 24.8104,C -3.1755,E1 25.1111,E2 135.8079} C_DIS
LIN {X 6.4182,Y -7.9874,Z 53,A -60.4419,B 24.8123,C -3.1598,E1 25.0965,E2 142.6555} C_DIS
LIN {X 5.606,Y -8.5773,Z 53,A -65.7344,B 24.8134,C -3.1505,E1 25.0843,E2 147.9519} C_DIS
LIN {X 4.6155,Y -9.1474,Z 53,A -72.8951,B 24.8151,C -3.1362,E1 25.0667,E2 155.1264} C_DIS
LIN {X 3.7328,Y -9.5425,Z 53,A -77.9077,B 24.8157,C -3.1305,E1 25.0537,E2 160.141} C_DIS
LIN {X 2.4048,Y -9.9601,Z 53,A -85.1466,B 24.8164,C -3.1246,E1 25.0343,E2 167.3818} C_DIS
LIN {X 0.914,Y -10.2059,Z 53,A -95.3866,B 24.8178,C -3.1126,E1 25.0059,E2 177.6424} C_DIS
LIN {X 0.914,Y -10.2059,Z 53,A -95.3866,B 24.8178,C -3.1126,E1 25.0059,E2 177.6424} C_DIS
Enddeposition()
LIN {X 0.0583,Y -11.1487,Z 53,A -97.7249,B 24.8188,C -3.1042,E1 24.9993,E2 180.0005} C_DIS
Startdeposition()
$VEL.CP = VEL_PRINT
LIN {X 0.8357,Y -11.1195,Z 53,A -91.6026,B 24.8177,C -3.1142,E1 25.0164,E2 173.8563} C_DIS
LIN {X 2.1689,Y -10.9356,Z 53,A -86.0986,B 24.8178,C -3.1128,E1 25.0316,E2 168.3607} C_DIS
LIN {X 2.9803,Y -10.746,Z 53,A -80.5127,B 24.8166,C -3.123,E1 25.0468,E2 162.7589} C_DIS
LIN {X 4.0962,Y -10.3727,Z 53,A -74.5782,B 24.8158,C -3.1301,E1 25.0623,E2 156.8197} C_DIS
LIN {X 4.9808,Y -9.9766,Z 53,A -69.3402,B 24.8147,C -3.1392,E1 25.0756,E2 151.5739} C_DIS
LIN {X 6.1194,Y -9.3233,Z 53,A -62.9063,B 24.8135,C -3.1496,E1 25.0909,E2 145.1353} C_DIS
LIN {X 7.0516,Y -8.6398,Z 53,A -56.6151,B 24.8118,C -3.164,E1 25.1048,E2 138.8331} C_DIS
LIN {X 8.0552,Y -7.7085,Z 53,A -51.2035,B 24.811,C -3.1705,E1 25.1157,E2 133.4284} C_DIS
LIN {X 8.6592,Y -7.0278,Z 53,A -45.3199,B 24.8087,C -3.1896,E1 25.1265,E2 127.5262} C_DIS
LIN {X 9.3158,Y -6.1308,Z 53,A -39.6024,B 24.8068,C -3.2049,E1 25.1356,E2 121.8003} C_DIS
LIN {X 9.8991,Y -5.136,Z 53,A -33.7499,B 24.8049,C -3.2211,E1 25.1436,E2 115.9399} C_DIS
LIN {X 10.3602,Y -4.1276,Z 53,A -28.0956,B 24.8029,C -3.2376,E1 25.1498,E2 110.2775} C_DIS
LIN {X 10.6883,Y -3.1799,Z 53,A -22.6002,B 24.8007,C -3.2555,E1 25.1545,E2 104.7709} C_DIS
LIN {X 10.9901,Y -1.8879,Z 53,A -16.1271,B 24.7983,C -3.2741,E1 25.1581,E2 98.2913} C_DIS
LIN {X 11.1317,Y -0.6546,Z 53,A -9.8068,B 24.7959,C -3.2936,E1 25.1597,E2 91.9624} C_DIS
LIN {X 11.1475,Y 0.2621,Z 53,A -5.09,B 24.7941,C -3.3082,E1 25.1596,E2 87.2389} C_DIS
LIN {X 11.0564,Y 1.4569,Z 53,A 0.9261,B 24.7919,C -3.3261,E1 25.1579,E2 81.216} C_DIS
LIN {X 10.8719,Y 2.4832,Z 53,A 6.2694,B 24.7898,C -3.3421,E1 25.1549,E2 75.866} C_DIS
LIN {X 10.5906,Y 3.4923,Z 53,A 11.9333,B 24.7876,C -3.3596,E1 25.1503,E2 70.1928} C_DIS
LIN {X 10.1181,Y 4.689,Z 53,A 18.0609,B 24.7857,C -3.3748,E1 25.1436,E2 64.0628} C_DIS
LIN {X 9.6709,Y 5.5532,Z 53,A 23.5672,B 24.7836,C -3.391,E1 25.1361,E2 58.5466} C_DIS
LIN {X 8.9525,Y 6.6492,Z 53,A 29.7164,B 24.782,C -3.4038,E1 25.1264,E2 52.3972} C_DIS
LIN {X 8.3351,Y 7.4088,Z 53,A 35.2038,B 24.7802,C -3.4177,E1 25.1164,E2 46.9017} C_DIS
LIN {X 7.5234,Y 8.2318,Z 53,A 41.0108,B 24.7787,C -3.4288,E1 25.1047,E2 41.0923} C_DIS
LIN {X 6.6654,Y 8.9401,Z 53,A 46.5805,B 24.7775,C -3.4381,E1 25.0924,E2 35.5213} C_DIS
LIN {X 5.7728,Y 9.5399,Z 53,A 52.1194,B 24.7764,C -3.4464,E1 25.0794,E2 29.9803} C_DIS
LIN {X 4.7942,Y 10.0672,Z 53,A 57.9181,B 24.7755,C -3.4538,E1 25.0649,E2 24.1799} C_DIS
LIN {X 3.6982,Y 10.5202,Z 53,A 64.0817,B 24.7747,C -3.4597,E1 25.0488,E2 18.0154} C_DIS
LIN {X 2.3429,Y 10.9004,Z 53,A 69.7009,B 24.775,C -3.4573,E1 25.0337,E2 12.4109} C_DIS
LIN {X 1.4446,Y 11.0579,Z 53,A 76.0398,B 24.774,C -3.4651,E1 25.0162,E2 6.0595} C_DIS
LIN {X 0.326,Y 11.1461,Z 53,A 81.8078,B 24.774,C -3.4649,E1 25.0001,E2 0.2939} C_DIS
LIN {X -0.8297,Y 11.1199,Z 53,A 87.5455,B 24.7744,C -3.4622,E1 24.9841,E2 -5.4387} C_DIS
LIN {X -2.1739,Y 10.9346,Z 53,A 93.1099,B 24.7755,C -3.4535,E1 24.9688,E2 -10.9872} C_DIS
LIN {X -3.0601,Y 10.7241,Z 53,A 99.3633,B 24.7755,C -3.4531,E1 24.9519,E2 -17.2488} C_DIS
LIN {X -4.3396,Y 10.2702,Z 53,A 106.0552,B 24.7768,C -3.4435,E1 24.9345,E2 -23.932} C_DIS
LIN {X -5.5309,Y 9.6833,Z 53,A 113.3195,B 24.7781,C -3.4334,E1 24.9166,E2 -31.192} C_DIS
LIN {X -6.5258,Y 9.0433,Z 53,A 119.3948,B 24.7797,C -3.4217,E1 24.9026,E2 -37.26} C_DIS
LIN {X -7.5253,Y 8.23,Z 53,A 125.5653,B 24.7816,C -3.4067,E1 24.8895,E2 -43.4186} C_DIS
Enddeposition()
END
